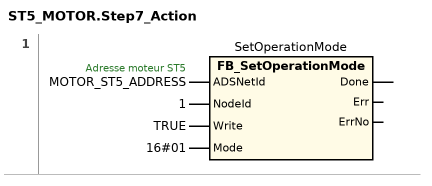
// NETWORK 1
//   MOTOR_ST5_ADDRESS: Adresse moteur ST5
SetOperationMode(ADSNetId := MOTOR_ST5_ADDRESS, NodeId := 1, Write := TRUE, Mode := 16#01); // FB_SetOperationMode
END_ACTION

END_PROGRAM

// ---- POUs/STATIONS/ST1_HT.TcPOU
PROGRAM ST1_HT
VAR
	STEP: INT := 0;
	START_TAMPO_AIR: BOOL;
	TAMPO_AIR: TON;
	JIG_STATUS_R_TRIG: R_TRIG;
	START_TAMPO_CTRLIN: BOOL;
	TAMPO_CTRLIN_TP: TP;
	asdf: TP;
	TAMPO_LIBERATION_TON: TON;
	START_TAMPO_LIBERATION: BOOL;
	TAMPO_SORTIE_VERIN_HAUT_TON: TON;
	START_TAMPO_VERIN_HAUT: BOOL;
	TAMPO_SORTIE_VERIN_ELEC_TON: TON;
	START_TAMPO_VERIN_ELEC: BOOL;
END_VAR

(*******************************************************
*
* Station 1 - Haute Tension
*
*
*********************************************************)
IF NOT(GEMMA.STEP='F1') THEN
	STEP:=0;
END_IF;


CASE STEP OF

0: (*Init*)

	ST1_1V4 := FALSE;
	ST1_1V5 := FALSE;
	
	(*ST1_HT_CTRLIN 	:=FALSE;	(*Prise de contrôle par le PLC*)*)
	ST1_HT_TYPW 	:=FALSE;	(*Type de mesure FALSE: Rigidité dielectrique TRUE:Megomètre*)
	ST1_HT_N0		:=FALSE;	(*Numéro de programme*)
	ST1_HT_N1 		:=FALSE;	(*Numéro de programme*)
	ST1_HT_N2 		:=FALSE;	(*Numéro de programme*)
	ST1_HT_MES_DCH 	:=FALSE;	(*Passage en mesure / décharge FALSE: Décharge TRUE:Mesure*)
	
	FLAGS.ST1_RELEASE_CARRIER := FALSE;
	START_TAMPO_CTRLIN := FALSE;
	START_TAMPO_LIBERATION := FALSE;
	START_TAMPO_VERIN_HAUT := FALSE;
	START_TAMPO_VERIN_ELEC := FALSE;
	
	STEP := STEP + 10;
	
10: (*Attend une palette / flanc montant du status*)

	IF JIG_STATUS_R_TRIG.Q THEN
		STEP := STEP + 10;
	END_IF;
	
20: (*Descend le vérin du dessus*)

	ST1_1V4 := TRUE;
	START_TAMPO_VERIN_HAUT := TRUE;
	STEP := STEP + 10;
	
30: (*Attend vérin dessus sorti*)

	IF TAMPO_SORTIE_VERIN_HAUT_TON.Q THEN
		START_TAMPO_VERIN_HAUT := FALSE;
		STEP := STEP + 10;
	END_IF;

40: (*Sort le vérin électrique*)

	ST1_1V5 := TRUE;
	START_TAMPO_VERIN_ELEC := TRUE;
	STEP := STEP + 10;
	
50: (*Attend vérin électrique sortie*)

	IF TAMPO_SORTIE_VERIN_ELEC_TON.Q THEN
		START_TAMPO_VERIN_ELEC := FALSE;
		STEP := 100;
	END_IF;

	
(**************************************************************************)
100: (*ACtive la prise en main de HT par le PLC et charge le programme*)

	ST1_HT_CTRLIN 	:= TRUE; 	(*active la communication API vers HT*)
	ST1_HT_TYPW 	:= FALSE;	(*Type de mesure FALSE: Rigidité dielectrique TRUE:Megomètre*)
	ST1_HT_N0		:= GETBIT32(inVal32:= INT_TO_DWORD(PUMP_PARAMS.ST1_HT_NO_PROG), bitNo:=0 ) ;	(*Numéro de programme bit 0*)
	ST1_HT_N1 		:= GETBIT32(inVal32:= INT_TO_DWORD(PUMP_PARAMS.ST1_HT_NO_PROG), bitNo:=1 ) ;	(*Numéro de programme bit 1*)
	ST1_HT_N2 		:= GETBIT32(inVal32:= INT_TO_DWORD(PUMP_PARAMS.ST1_HT_NO_PROG), bitNo:=2 ) ;	(*Numéro de programme bit 2*)
	
	STEP := STEP + 10;

110: (*Démarre la mesure*)

	ST1_HT_MES_DCH 	:=TRUE;	(*Passage en mesure / décharge FALSE: Décharge TRUE:Mesure*)
	
	STEP := STEP + 10;	

120: (*Attend début du test HT*)

	IF NOT(ST1_HT_EOT) THEN
		STEP := STEP + 10;
	END_IF;

130: (*Attend la fin du test HT*)

	IF ST1_HT_EOT THEN
		ST1_HT_OK := ST1_HT_PASS;
		STEP := STEP + 10;
	END_IF;
	
140: (*Termine le test*)

	ST1_HT_MES_DCH 	:=FALSE;	(*Passage en mesure / décharge FALSE: Décharge TRUE:Mesure*)
	
	STEP := 300;	

(**************************************************************************)	

300: (*Rentre le vérin électrique*)

	ST1_1V5 := FALSE;
	STEP := STEP + 10;
	
310: (*Monte le vérin du dessus*)

	ST1_1V4 := FALSE;
	STEP := STEP + 10;

320: (*Libère la palette*)
	
	FLAGS.ST1_RELEASE_CARRIER := TRUE;
	STEP := 0;


ELSE
    (*default case*);
END_CASE;

(*FBs*)
TAMPO_SORTIE_VERIN_HAUT_TON(IN:= START_TAMPO_VERIN_HAUT, PT:= TEMPS_SORTIE_VERIN);
TAMPO_SORTIE_VERIN_ELEC_TON(IN:= START_TAMPO_VERIN_ELEC, PT:= TEMPS_SORTIE_VERIN);

TAMPO_CTRLIN_TP(IN:= START_TAMPO_CTRLIN, PT:= T#1S);
TAMPO_LIBERATION_TON(IN:= START_TAMPO_LIBERATION, PT:= T#1S);
JIG_STATUS_R_TRIG(CLK:= CONVEYOR.JIG_ST1.STATUS);
PROG_STEPS.ST1:=STEP;

END_PROGRAM

// ---- POUs/STATIONS/ST2_ASPIRATION.TcPOU
PROGRAM ST2_ASPIRATION
VAR
	STEP: INT := 0;
	JIG_STATUS_R_TRIG: R_TRIG;
	TAMPO_AMORCAGE_TON: TON;
	START_TAMPO_AMORCAGE: BOOL;
	TAMPO_MESURE_TON: TON;
	START_TAMPO_MESURE: BOOL;
	TAMPO_SORTIE_VERIN_HAUT_TON: TON;
	START_TAMPO_VERIN_HAUT: BOOL;
	TAMPO_SORTIE_VERIN_BAS_TON: TON;
	START_TAMPO_VERIN_BAS: BOOL;
	TAMPO_SORTIE_VERIN_ELEC_TON: TON;
	START_TAMPO_VERIN_ELEC: BOOL;
	START_TAMPO_MESURE_PERTES: BOOL;
	TAMPO_MESURE_PERTES_TON: TON;
END_VAR

(*******************************************************
*
* Station 2 - Aspiration
*
*
*********************************************************)
IF NOT(GEMMA.STEP='F1') THEN
	STEP:=0;
END_IF;


CASE STEP OF

0: (*Init*)

	ST2_2V4 := FALSE;
	ST2_2V5 := FALSE;
	ST2_2V6 := FALSE;
	ST2_2V7 := FALSE;
	ST2_2V8 := FALSE;
	
	FLAGS.ST2_RELEASE_CARRIER := FALSE;
	START_TAMPO_AMORCAGE := FALSE;
	START_TAMPO_MESURE := FALSE;
	START_TAMPO_VERIN_ELEC := FALSE;
	START_TAMPO_VERIN_HAUT := FALSE;
	START_TAMPO_VERIN_BAS := FALSE;
	
	STEP := STEP + 10;
	
10: (*Attend une palette / flanc montant du status*)

	IF JIG_STATUS_R_TRIG.Q THEN
		STEP := STEP + 10;
	END_IF;
	
20: (*Descend le vérin du dessus*)

	ST2_2V4 := TRUE;
	START_TAMPO_VERIN_HAUT := TRUE;
	STEP := STEP + 10;
	
30: (*Attend vérin dessus sorti*)

	IF TAMPO_SORTIE_VERIN_HAUT_TON.Q THEN
		START_TAMPO_VERIN_HAUT := FALSE;
		STEP := STEP + 10;
	END_IF;

40: (*Monte le vérin du dessous*)

	ST2_2V5 := TRUE;
	START_TAMPO_VERIN_BAS := TRUE;
	STEP := STEP + 10;
	
50: (*Attend vérin dessus sorti*)

	IF TAMPO_SORTIE_VERIN_BAS_TON.Q THEN
		START_TAMPO_VERIN_BAS := FALSE;
		STEP := STEP + 10;
	END_IF;
	
60: (*Sort le vérin électrique*)

	ST2_2V6 := TRUE;
	IF PUMP_PARAMS.GEN_BYPASS THEN
		ST2_2V7 := TRUE;
	END_IF
	START_TAMPO_VERIN_ELEC := TRUE;
	STEP := STEP + 10;
	
70: (*Attend vérin électrique sortie*)

	IF TAMPO_SORTIE_VERIN_ELEC_TON.Q THEN
		START_TAMPO_VERIN_ELEC := FALSE;
		STEP := STEP + 10;
	END_IF;

80: (*Allume la pompe*)

	IF PUMP_PARAMS.ST2_CONTRE_PRESSION THEN (*ouvre la vanne de contre pression d'air si nécessaire*)
		ST2_2V8:=TRUE;
	END_IF;
	
	ST2_POWER := TRUE;
	STEP := 100;
	
(**************************************************************************)
100: (*Démarre la tampo pour l'amorcage*)

	START_TAMPO_AMORCAGE := TRUE;
	STEP := STEP + 10;
	
110: (*Attend fin tampo amorcage*)

	IF TAMPO_AMORCAGE_TON.Q THEN
		START_TAMPO_AMORCAGE := FALSE;
		STEP := STEP + 10;
	END_IF;
	
120: (*Démarre la tampo pour la mesure de pression*)

	START_TAMPO_MESURE := TRUE;
	STEP := STEP + 10;
	
130: (*Attend fin tampo mesure - MESURE EN COURT*)

	IF TAMPO_MESURE_TON.Q THEN
		START_TAMPO_MESURE := FALSE;
		ST2_2V8:=FALSE; (*ferme la vanne de contre pression d'air*)
		STEP := STEP + 10;
	END_IF;
	
140: (*Démarre la tampo pour la mesure de la tenue aspiration*)

	START_TAMPO_MESURE_PERTES := TRUE;
	ST2_POWER := FALSE;
	STEP := STEP + 10;
	
150: (*Attend fin tampo mesure - MESURE EN COURT tenue aspiration*)

	IF TAMPO_MESURE_PERTES_TON.Q THEN
		START_TAMPO_MESURE_PERTES := FALSE;
		ST2_2V8:=FALSE; (*ferme la vanne de contre pression d'air*)
		STEP := 300;
	END_IF;
	

(**************************************************************************)	

300: (*Rentre le vérin électrique*)

	ST2_2V6 := FALSE;
	ST2_2V7 := TRUE;
	STEP := STEP + 10;
	
310: (*Descend le vérin du dessous*)

	ST2_2V5 := FALSE;
	STEP := STEP + 10;
	
320: (*Monte le vérin du dessus*)

	ST2_2V4 := FALSE;
	STEP := STEP + 10;

330: (*Libère la palette*)

	FLAGS.ST2_RELEASE_CARRIER := TRUE;
	STEP := 0;


ELSE
    (*default case*);
END_CASE;

(*FBs*)
TAMPO_SORTIE_VERIN_HAUT_TON(IN:= START_TAMPO_VERIN_HAUT, PT:= TEMPS_SORTIE_VERIN);
TAMPO_SORTIE_VERIN_BAS_TON(IN:= START_TAMPO_VERIN_BAS, PT:= TEMPS_SORTIE_VERIN);
TAMPO_SORTIE_VERIN_ELEC_TON(IN:= START_TAMPO_VERIN_ELEC, PT:= TEMPS_SORTIE_VERIN);

TAMPO_AMORCAGE_TON(IN:= START_TAMPO_AMORCAGE, PT:= PUMP_PARAMS.ST6_TEMPS_POMPAGE);
TAMPO_MESURE_TON(IN:= START_TAMPO_MESURE, PT:= PUMP_PARAMS.ST6_TEMPS_MESURE);
TAMPO_MESURE_PERTES_TON(IN:= START_TAMPO_MESURE_PERTES, PT:= PUMP_PARAMS.ST2_TEMPS_MESURE_PERTE_PRESSION);
JIG_STATUS_R_TRIG(CLK:= CONVEYOR.JIG_ST2.STATUS);
PROG_STEPS.ST2:=STEP;

END_PROGRAM

// ---- POUs/STATIONS/ST3_ETANCHEITE.TcPOU
PROGRAM ST3_ETANCHEITE
VAR
	STEP: INT := 0;
	JIG_STATUS_R_TRIG: R_TRIG;
	START_TAMPO_MISE_SOUS_PRESSION: BOOL;
	TAMPO_MISE_SOUS_PRESSION: TON;
	START_TAMPO_STABILISATION: BOOL;
	TAMPO_STABILISATION: TON;
	START_TAMPO_MESURE: BOOL;
	TAMPO_MESURE: TON;
	PRESSION_DEBUT: REAL;
	PRESSION_FIN: REAL;
	TAMPO_SORTIE_VERIN_HAUT_TON: TON;
	START_TAMPO_VERIN_HAUT: BOOL;
	TAMPO_SORTIE_VERIN_BAS_TON: TON;
	START_TAMPO_VERIN_BAS: BOOL;
	TAMPO_DEPRESSION_TON: TON;
	START_TAMPO_DEPRESSION: BOOL;
	PRESSION_DEBUT_ABS: REAL;
END_VAR

(*******************************************************
*
* Station 3 - Etanchéité
*
*
*********************************************************)
IF NOT(GEMMA.STEP='F1') THEN
	STEP:=0;
END_IF;


CASE STEP OF

0: (*Init*)

	ST3_3V4 := FALSE;
	ST3_3V5 := FALSE;
	ST3_3V10 := FALSE;
	ST3_3V11 := FALSE;
	ST3_3V12 := TRUE;
	
	FLAGS.ST3_RELEASE_CARRIER := FALSE;
	
	START_TAMPO_MISE_SOUS_PRESSION := FALSE;
	START_TAMPO_STABILISATION := FALSE;
	START_TAMPO_MESURE := FALSE;
	START_TAMPO_VERIN_HAUT := FALSE;
	START_TAMPO_VERIN_BAS := FALSE;
	START_TAMPO_DEPRESSION := FALSE;

	
	STEP := STEP + 10;
	
10: (*Attend une palette / flanc montant du status*)

	IF JIG_STATUS_R_TRIG.Q THEN
		STEP := STEP + 10;
	END_IF;
	
20: (*Descend le vérin du dessus*)

	ST3_3V4 := TRUE;
	START_TAMPO_VERIN_HAUT := TRUE;
	STEP := STEP + 10;
	
30: (*Attend vérin dessus sorti*)

	IF TAMPO_SORTIE_VERIN_HAUT_TON.Q THEN
		START_TAMPO_VERIN_HAUT :=FALSE;
		STEP := STEP + 10;
	END_IF;

40: (*Monte le vérin du dessous*)

	ST3_3V5 := TRUE;
	IF PUMP_PARAMS.GEN_BYPASS THEN
		ST3_3V7 := TRUE;
	END_IF
	START_TAMPO_VERIN_BAS := TRUE;
	STEP := STEP + 10;
	
50: (*Attend vérin dessus sorti*)

	IF TAMPO_SORTIE_VERIN_BAS_TON.Q THEN
		START_TAMPO_VERIN_BAS := FALSE;
		STEP := 100;
	END_IF;
	
	
(**************************************************************************)
100: (*Mise sous pression de la cartouche*)

	ST3_3V10 := TRUE;
	ST3_3V11 := FALSE;
	ST3_3V12 := TRUE;
	
	START_TAMPO_MISE_SOUS_PRESSION := TRUE;
	
	STEP := STEP + 10;
	
	
110: (*Tampo pour la mise sous pression de la cartouche*)

	IF TAMPO_MISE_SOUS_PRESSION.Q THEN
		START_TAMPO_MISE_SOUS_PRESSION := FALSE;
		STEP := STEP + 10;
	END_IF;

120: (*Start stabilisation*)

	START_TAMPO_STABILISATION := TRUE;
	ST3_3V10 := FALSE;
	
	STEP := STEP + 10;	

130: (*Tampo pour la stabilisation de la pression dans la cartouche*)

	IF TAMPO_STABILISATION.Q THEN
		START_TAMPO_STABILISATION := FALSE;
		STEP := STEP + 10;
	END_IF;
	
140: (*Start mesure*)

	START_TAMPO_MESURE := TRUE;
	ST3_3V12 := FALSE;
	PRESSION_DEBUT := ST3_PRESSION; (* Mesure de la pression différentielle au début du test *)
	
	STEP := STEP + 10;	

150: (*Tampo pour la mesure du delta P*)

	IF TAMPO_MESURE.Q THEN
		START_TAMPO_MESURE := FALSE;
		PRESSION_FIN := ST3_PRESSION; (* Mesure de la pression à la fin du test *)
		ST3_PRESSION_FIN_ABS := ST3_PRESSION_ABS; (* Mesure de la pression par rapport à l'atmosphère à la fin du test *)
		ST3_DELTA_P := PRESSION_FIN - PRESSION_DEBUT; (* Calcule de la chutte de pression *)
		STEP := STEP + 10;
	END_IF;
	
160: (*Fin mesure, dépressiorisation de la cartouche*)

	ST3_3V10 := FALSE;
	ST3_3V11 := TRUE;
	ST3_3V12 := TRUE;
	
	START_TAMPO_DEPRESSION := TRUE;
	
	STEP := STEP + 10;

170: (*Tampo dépression de cartouche*)

	IF TAMPO_DEPRESSION_TON.Q THEN
		START_TAMPO_DEPRESSION := FALSE;
		STEP := 300;
	END_IF;	
	
	

(**************************************************************************)	

300: (*Descend le vérin du dessous*)

	ST3_3V5 := FALSE;
	ST3_3V7 := FALSE;
	STEP := STEP + 10;
	
310: (*Monte le vérin du dessus*)

	ST3_3V4 := FALSE;
	STEP := STEP + 10;

320: (*Libère la palette*)

	FLAGS.ST3_RELEASE_CARRIER := TRUE;
	STEP := 0;


ELSE
    (*default case*);
END_CASE;

(*FBs*)

TAMPO_SORTIE_VERIN_HAUT_TON(IN:= START_TAMPO_VERIN_HAUT, PT:= TEMPS_SORTIE_VERIN);
TAMPO_SORTIE_VERIN_BAS_TON(IN:= START_TAMPO_VERIN_BAS, PT:= TEMPS_SORTIE_VERIN);

TAMPO_DEPRESSION_TON(IN:= START_TAMPO_DEPRESSION, PT:= T#2S);
TAMPO_MISE_SOUS_PRESSION(IN:= START_TAMPO_MISE_SOUS_PRESSION, PT:= PUMP_PARAMS.ST3_TEMPS_MISE_SOUS_PRESSION);
TAMPO_STABILISATION(IN:= START_TAMPO_STABILISATION, PT:= PUMP_PARAMS.ST3_TEMPS_STABILISATION);
TAMPO_MESURE(IN:= START_TAMPO_MESURE, PT:= PUMP_PARAMS.ST3_TEMPS_MESURE);
JIG_STATUS_R_TRIG(CLK:= CONVEYOR.JIG_ST3.STATUS);
PROG_STEPS.ST3:=STEP;

END_PROGRAM

// ---- POUs/STATIONS/ST4_DEBIT_PETIT.TcPOU
PROGRAM ST4_DEBIT_PETIT
VAR
	STEP: INT := 0;
	JIG_STATUS_R_TRIG: R_TRIG;
	START_TAMPO_AMORCAGE: BOOL;
	TAMPO_AMORCAGE_TON: TON;
	START_TAMPO_REGLAGE: BOOL;
	TAMPO_REGLAGE_TON: TON;
	START_TAMPO_MESURE_DEBIT: BOOL;
	TAMPO_MESURE_DEBIT_TON: TON;
	START_TAMPO_VIDANGE: BOOL;
	TAMPO_VIDANGE_TON: TON;
	START_TAMPO_MESURE_DEBIT_MAX: BOOL;
	TAMPO_MESURE_DEBIT_MAX_TON: TON;
	POIDS_QMAX_DEBUT: REAL;
	POIDS_Q_DEBUT: REAL;
	P_ERREUR: REAL;
	START_TAMPO_PRESSION: BOOL;
	TAMPO_PRESSION_TON: TON;
		TAMPO_SORTIE_VERIN_HAUT_TON: TON;
	START_TAMPO_VERIN_HAUT: BOOL;
	TAMPO_SORTIE_VERIN_BAS_TON: TON;
	START_TAMPO_VERIN_BAS: BOOL;
	TAMPO_SORTIE_VERIN_ELEC_TON: TON;
	START_TAMPO_VERIN_ELEC: BOOL;
END_VAR

(*******************************************************
*
* Station 4 - Petits débits
*
*
*********************************************************)
IF NOT(GEMMA.STEP='F1') THEN
	STEP:=0;
END_IF;


CASE STEP OF

0: (*Init*)

	ST4_4V4 := FALSE;
	ST4_4V5 := FALSE;
	ST4_4V6 := FALSE;
	ST4_4V7 := FALSE;

	ST4_4V10 := FALSE;
	ST4_4V12 := FALSE;
	ST4_4V13 := FALSE;
	
	
	FLAGS.ST4_RELEASE_CARRIER := FALSE;
	START_TAMPO_AMORCAGE := FALSE;
	START_TAMPO_MESURE_DEBIT:= FALSE;
	START_TAMPO_MESURE_DEBIT_MAX:= FALSE;
	START_TAMPO_VIDANGE:= FALSE;
	START_TAMPO_REGLAGE:= FALSE;
	START_TAMPO_PRESSION:= FALSE;
	START_TAMPO_VERIN_ELEC := FALSE;
	START_TAMPO_VERIN_HAUT := FALSE;
	START_TAMPO_VERIN_BAS := FALSE;
	
	
	STEP := STEP + 10;
	
10: (*Attend une palette / flanc montant du status*)

	IF JIG_STATUS_R_TRIG.Q THEN
		STEP := STEP + 10;
	END_IF;
	
20: (*Descend le vérin du dessus*)

	ST4_4V4 := TRUE;
	START_TAMPO_VERIN_HAUT := TRUE;
	POIDS_QMAX_DEBUT	:= 0;	(*Met à 0 les différentes variables pour le calcul et résultat des débits*)
	POIDS_Q_DEBUT		:= 0;
	ST4_Q				:= 0;
	ST4_QMAX			:= 0;
	STEP := STEP + 10;
	
30: (*Attend vérin dessus sorti*)

	IF TAMPO_SORTIE_VERIN_HAUT_TON.Q THEN
		START_TAMPO_VERIN_HAUT := FALSE;
		STEP := STEP + 10;
	END_IF;

40: (*Monte le vérin du dessous*)

	ST4_4V5 := TRUE;
	START_TAMPO_VERIN_BAS := TRUE;
	STEP := STEP + 10;
	
50: (*Attend vérin dessus sorti*)

	IF TAMPO_SORTIE_VERIN_BAS_TON.Q THEN
		START_TAMPO_VERIN_BAS := FALSE;
		STEP := STEP + 10;
	END_IF;
	
60: (*Sort le vérin électrique*)

	ST4_4V6 := TRUE;
	IF PUMP_PARAMS.GEN_BYPASS THEN
		ST4_4V7 := TRUE;
	END_IF
	START_TAMPO_VERIN_ELEC := TRUE;
	STEP := STEP + 10;
	
70: (*Attend vérin électrique sortie*)

	IF TAMPO_SORTIE_VERIN_ELEC_TON.Q THEN
		START_TAMPO_VERIN_ELEC := FALSE;
		STEP := STEP + 10;
	END_IF;
	
80: (*Si la balance est trop pleine, attend qu'elle soit vidée suffisament avant d'allumer la pompe*)
	
	IF ST4_POIDS<BALANCE_POIDS_LIMITE THEN
		STEP:=STEP + 10;
	END_IF
		
90: (*Allume la pompe*)

	ST4_POWER := TRUE;
	ST4_4V10 := TRUE;
	ST4_4V13 := TRUE;
	STEP := 100;
	
	
(**************************************************************************)
100: (*Démarre la tampo pour l'amorcage*)

	START_TAMPO_AMORCAGE := TRUE;
	STEP := STEP + 10;
	
110: (*Attend fin tampo amorcage*)

	IF TAMPO_AMORCAGE_TON.Q THEN
		START_TAMPO_AMORCAGE := FALSE;
		STEP := STEP + 10;
	END_IF;
	
120: (*Démarre la tampo pour la mesure de Qmax*)

	START_TAMPO_MESURE_DEBIT_MAX := TRUE;
	POIDS_QMAX_DEBUT := ST4_POIDS;
	STEP := STEP + 10;
	
130: (*Attend fin tampo mesure de Qmax ***********************************************************)
	IF TAMPO_MESURE_DEBIT_MAX_TON.Q THEN
		ST4_QMAX := CONVERT_MASS_TO_FLOW(ST4_POIDS - POIDS_QMAX_DEBUT, PUMP_PARAMS.ST45_TEMPS_MESURE_DEBIT_MAX);(*Calcul du débit max*)
		
		QMAX_ARRAY[INDEX_QMAX_ARRAY]:=ST4_QMAX; (*Array des derniers résultats*)
		INDEX_QMAX_ARRAY := INDEX_QMAX_ARRAY+1;
		
		START_TAMPO_MESURE_DEBIT_MAX := FALSE;
		ST4_4V12 := TRUE;
		ST4_4V13 := FALSE;
		STEP := STEP + 10;
	END_IF;
	
140: (*Démarre la tampo pour la mise sous pression*)

	START_TAMPO_PRESSION := TRUE;
	STEP := STEP + 10;
	
150: (*Attend fin tampo mise sous pression*)

	IF TAMPO_PRESSION_TON.Q THEN
		START_TAMPO_PRESSION := FALSE;
		STEP := STEP + 10;
	END_IF;
	
160: (*Démarre la tampo pour le réglage*)

	START_TAMPO_REGLAGE := TRUE;
	STEP := STEP + 10;
	
170: (*Attend fin tampo réglage*)

(*Réglage pression**********************************************)
PRESSURE_REGULATOR_ST4(
GEMMA				:= GEMMA.STEP,
COURANT				:= ST4_COURANT, 
PRESSION_CONSIGNE	:= PUMP_PARAMS.ST45_PRESSION_CONSIGNE, 
PRESSION_MESURE		:= ST4_PRESSURE_FILTERED,
MOTOR_POSITION_MAX	:= MOTOR_ST4_POSITION_MAX,
MOTOR_INITIAL_POSITION := MOTOR_ST4_INITIAL_POS,
MOTOR_POSITION		=> FLAGS.MOTOR_ST4_POSITION
);
	

	IF TAMPO_REGLAGE_TON.Q THEN
		START_TAMPO_REGLAGE := FALSE;
		STEP := STEP + 10;
	END_IF;
	
180: (*Démarre la tampo pour la mesure de debit*************************************************)

	START_TAMPO_MESURE_DEBIT := TRUE;
	POIDS_Q_DEBUT := ST4_POIDS;
	STEP := STEP + 10;

	
190: (*Attend fin tampo amorcage - MESURE EN COURT*)

(*Réglage pression***********************************************)
PRESSURE_REGULATOR_ST4( 
GEMMA				:= GEMMA.STEP,
COURANT				:= ST4_COURANT, 
PRESSION_CONSIGNE	:= PUMP_PARAMS.ST45_PRESSION_CONSIGNE, 
PRESSION_MESURE		:= ST4_PRESSURE_FILTERED,
MOTOR_POSITION_MAX	:= MOTOR_ST4_POSITION_MAX,
MOTOR_INITIAL_POSITION := MOTOR_ST4_INITIAL_POS,
MOTOR_POSITION		=> FLAGS.MOTOR_ST4_POSITION
);

	IF TAMPO_MESURE_DEBIT_TON.Q THEN
		ST4_Q := CONVERT_MASS_TO_FLOW(ST4_POIDS - POIDS_Q_DEBUT, PUMP_PARAMS.ST45_TEMPS_MESURE_DEBIT);(*Calcul du débit de travail*)
		
		Q_ARRAY[INDEX_Q_ARRAY]:=ST4_Q; (*Array des derniers résultats*)
		INDEX_Q_ARRAY := INDEX_Q_ARRAY+1;
		
		START_TAMPO_MESURE_DEBIT := FALSE;
		STEP := 300;
	END_IF;
	
	

(**************************************************************************)	

300: (*Descend le vérin du dessous*)

	ST4_4V5 := FALSE;
	ST4_4V10 := FALSE;	(* ferme la vanne avant la pompe*)
	ST4_4V12 := FALSE;
	ST4_4V13 := TRUE;
	STEP := STEP + 10;

310: (*Démarre la tampo de vidange de la pompe*)

	START_TAMPO_VIDANGE := TRUE;
	STEP := STEP + 10;
	
320: (*Attend fin tampo amorcage*)

	IF TAMPO_VIDANGE_TON.Q THEN
		START_TAMPO_VIDANGE := FALSE;
		ST4_4V13 := FALSE;
		ST4_POWER := FALSE;
		STEP := STEP + 10;
	END_IF;

330: (*Rentre le vérin électrique*)

	ST4_4V6 := FALSE;
	ST4_4V7 := FALSE;
	STEP := STEP + 10;
	
	
340: (*Monte le vérin du dessus*)

	ST4_4V4 := FALSE;
	STEP := STEP + 10;

350: (*Libère la palette*)

	FLAGS.ST4_RELEASE_CARRIER := TRUE;
	STEP := 0;


ELSE
    (*default case*);
END_CASE;

(*FBs*)
TAMPO_SORTIE_VERIN_HAUT_TON(IN:= START_TAMPO_VERIN_HAUT, PT:= TEMPS_SORTIE_VERIN);
TAMPO_SORTIE_VERIN_BAS_TON(IN:= START_TAMPO_VERIN_BAS, PT:= TEMPS_SORTIE_VERIN);
TAMPO_SORTIE_VERIN_ELEC_TON(IN:= START_TAMPO_VERIN_ELEC, PT:= TEMPS_SORTIE_VERIN);

TAMPO_AMORCAGE_TON(IN:= START_TAMPO_AMORCAGE, PT:= PUMP_PARAMS.ST45_TEMPS_POMPAGE);
TAMPO_REGLAGE_TON(IN:= START_TAMPO_REGLAGE, PT:= PUMP_PARAMS.ST45_TEMPS_REGLAGE_PRESSION);
TAMPO_VIDANGE_TON(IN:= START_TAMPO_VIDANGE, PT:= TEMPS_VIDANGE_POMPE);
TAMPO_PRESSION_TON(IN:= START_TAMPO_PRESSION, PT:= TEMPS_CHANGEMENT_PRESSION);
TAMPO_MESURE_DEBIT_TON(IN:= START_TAMPO_MESURE_DEBIT, PT:= PUMP_PARAMS.ST45_TEMPS_MESURE_DEBIT);
TAMPO_MESURE_DEBIT_MAX_TON(IN:= START_TAMPO_MESURE_DEBIT_MAX, PT:= PUMP_PARAMS.ST45_TEMPS_MESURE_DEBIT_MAX);
JIG_STATUS_R_TRIG(CLK:= CONVEYOR.JIG_ST4.STATUS);
PROG_STEPS.ST4:=STEP;

END_PROGRAM

// ---- POUs/Functions/CONVERT_MASS_TO_FLOW.TcPOU
FUNCTION CONVERT_MASS_TO_FLOW : REAL
VAR_INPUT
	Mass:REAL; (*in gramme*)
	Delay:TIME; (*in ms*)
END_VAR
VAR
END_VAR

CONVERT_MASS_TO_FLOW:=Mass/TIME_TO_DWORD(Delay)*60*60;

END_FUNCTION

// ---- POUs/STATIONS/ST5_GRAND_PETIT.TcPOU
PROGRAM ST5_GRAND_PETIT
VAR
	STEP: INT := 0;
	JIG_STATUS_R_TRIG: R_TRIG;
	START_TAMPO_AMORCAGE: BOOL;
	TAMPO_AMORCAGE_TON: TON;
	START_TAMPO_REGLAGE: BOOL;
	TAMPO_REGLAGE_TON: TON;
	START_TAMPO_MESURE_DEBIT: BOOL;
	TAMPO_MESURE_DEBIT_TON: TON;
	START_TAMPO_VIDANGE: BOOL;
	TAMPO_VIDANGE_TON: TON;
	START_TAMPO_MESURE_DEBIT_MAX: BOOL;
	TAMPO_MESURE_DEBIT_MAX_TON: TON;
	POIDS_QMAX_DEBUT: REAL;
	POIDS_Q_DEBUT: REAL;
	P_ERREUR: REAL;
	START_TAMPO_PRESSION: BOOL;
	TAMPO_PRESSION_TON: TON;
	TAMPO_SORTIE_VERIN_HAUT_TON: TON;
	START_TAMPO_VERIN_HAUT: BOOL;
	TAMPO_SORTIE_VERIN_BAS_TON: TON;
	START_TAMPO_VERIN_BAS: BOOL;
	TAMPO_SORTIE_VERIN_ELEC_TON: TON;
	START_TAMPO_VERIN_ELEC: BOOL;
	TAMPO_RENTREE_VERIN_HAUT_TON: TON;
	START_TAMPO_RENTREE_VERIN_HAUT: BOOL;
END_VAR

(*******************************************************
*
* Station 5 - Grands débits
*
*
*********************************************************)
IF NOT(GEMMA.STEP='F1') THEN
	STEP:=0;
END_IF;


CASE STEP OF

0: (*Init*)

	ST5_5V4 := FALSE;
	ST5_5V5 := FALSE;
	ST5_5V6 := FALSE;

	ST5_5V10 := FALSE;
	ST5_5V12 := FALSE;
	ST5_5V13 := FALSE;
	
	
	FLAGS.ST5_RELEASE_CARRIER := FALSE;
	START_TAMPO_AMORCAGE := FALSE;
	START_TAMPO_MESURE_DEBIT:= FALSE;
	START_TAMPO_MESURE_DEBIT_MAX:= FALSE;
	START_TAMPO_VIDANGE:= FALSE;
	START_TAMPO_REGLAGE:= FALSE;
	START_TAMPO_PRESSION:= FALSE;
	START_TAMPO_VERIN_ELEC := FALSE;
	START_TAMPO_VERIN_HAUT := FALSE;
	START_TAMPO_VERIN_BAS := FALSE;
	
	
	STEP := STEP + 10;
	
10: (*Attend une palette / flanc montant du status*)

	IF JIG_STATUS_R_TRIG.Q THEN
		STEP := STEP + 10;
	END_IF;
	
20: (*Descend le vérin du dessus*)

	ST5_5V4 := TRUE;
	START_TAMPO_VERIN_HAUT := TRUE;
	POIDS_QMAX_DEBUT	:= 0;	(*Met à 0 les différentes variables pour le calcul et résultat des débits*)
	POIDS_Q_DEBUT		:= 0;
	ST5_Q				:= 0;
	ST5_QMAX			:= 0;
	STEP := STEP + 10;
	
30: (*Attend vérin dessus sorti*)

	IF TAMPO_SORTIE_VERIN_HAUT_TON.Q THEN
		START_TAMPO_VERIN_HAUT := FALSE;
		STEP := STEP + 10;
	END_IF;

40: (*Monte le vérin du dessous*)

	ST5_5V5 := TRUE;
	START_TAMPO_VERIN_BAS := TRUE;
	STEP := STEP + 10;
	
50: (*Attend vérin dessus sorti*)

	IF TAMPO_SORTIE_VERIN_BAS_TON.Q THEN
		START_TAMPO_VERIN_BAS := FALSE;
		STEP := STEP + 10;
	END_IF;
	
60: (*Sort le vérin électrique*)

	ST5_5V6 := TRUE;
	START_TAMPO_VERIN_ELEC := TRUE;
	STEP := STEP + 10;
	
70: (*Attend vérin électrique sortie*)

	IF TAMPO_SORTIE_VERIN_ELEC_TON.Q THEN
		START_TAMPO_VERIN_ELEC := FALSE;
		STEP := STEP + 10;
	END_IF;

80: (*Si la balance est trop pleine, attend qu'elle soit vidée suffisament avant d'allumer la pompe*)
	
IF ST5_POIDS<BALANCE_POIDS_LIMITE THEN
	STEP:=STEP + 10;
END_IF
	
90: (*Allume la pompe*)

	ST5_POWER := TRUE;
	ST5_5V10 := TRUE;
	ST5_5V13 := TRUE;
	STEP := 100;
	
	
(**************************************************************************)
100: (*Démarre la tampo pour l'amorcage*)

	START_TAMPO_AMORCAGE := TRUE;
	STEP := STEP + 10;
	
110: (*Attend fin tampo amorcage*)

	IF TAMPO_AMORCAGE_TON.Q THEN
		START_TAMPO_AMORCAGE := FALSE;
		STEP := STEP + 10;
	END_IF;
	
120: (*Démarre la tampo pour la mesure de Qmax*)

	START_TAMPO_MESURE_DEBIT_MAX := TRUE;
	POIDS_QMAX_DEBUT := ST5_POIDS;
	STEP := STEP + 10;
	
130: (*Attend fin tampo mesure de Qmax ***********************************************************)
	IF TAMPO_MESURE_DEBIT_MAX_TON.Q THEN
		ST5_QMAX := CONVERT_MASS_TO_FLOW(ST5_POIDS - POIDS_QMAX_DEBUT, PUMP_PARAMS.ST45_TEMPS_MESURE_DEBIT_MAX);(*Calcul du débit max*)
		
		QMAX5_ARRAY[INDEX_QMAX5_ARRAY]:=ST5_QMAX; (*Array des derniers résultats*)
		INDEX_QMAX5_ARRAY := INDEX_QMAX5_ARRAY+1;
		
		START_TAMPO_MESURE_DEBIT_MAX := FALSE;
		ST5_5V12 := TRUE;
		ST5_5V13 := FALSE;
		STEP := STEP + 10;
	END_IF;
	
140: (*Démarre la tampo pour la mise sous pression*)

	START_TAMPO_PRESSION := TRUE;
	STEP := STEP + 10;
	
150: (*Attend fin tampo mise sous pression*)

	IF TAMPO_PRESSION_TON.Q THEN
		START_TAMPO_PRESSION := FALSE;
		STEP := STEP + 10;
	END_IF;
	
160: (*Démarre la tampo pour le réglage*)

	START_TAMPO_REGLAGE := TRUE;
	STEP := STEP + 10;
	
170: (*Attend fin tampo réglage*)

(*Réglage pression**********************************************)
PRESSURE_REGULATOR_ST5(
GEMMA				:= GEMMA.STEP,
COURANT				:= ST5_COURANT, 
PRESSION_CONSIGNE	:= PUMP_PARAMS.ST45_PRESSION_CONSIGNE, 
PRESSION_MESURE		:= ST5_PRESSURE_FILTERED,
MOTOR_POSITION_MAX	:= MOTOR_ST5_POSITION_MAX,
MOTOR_INITIAL_POSITION := MOTOR_ST5_INITIAL_POS,
MOTOR_POSITION		=> FLAGS.MOTOR_ST5_POSITION
);
	

	IF TAMPO_REGLAGE_TON.Q THEN
		START_TAMPO_REGLAGE := FALSE;
		STEP := STEP + 10;
	END_IF;
	
180: (*Démarre la tampo pour la mesure de debit*************************************************)

	START_TAMPO_MESURE_DEBIT := TRUE;
	POIDS_Q_DEBUT := ST5_POIDS;
	STEP := STEP + 10;

	
190: (*Attend fin tampo amorcage - MESURE EN COURT*)

(*Réglage pression***********************************************)
PRESSURE_REGULATOR_ST5( 
GEMMA				:= GEMMA.STEP,
COURANT				:= ST5_COURANT, 
PRESSION_CONSIGNE	:= PUMP_PARAMS.ST45_PRESSION_CONSIGNE, 
PRESSION_MESURE		:= ST5_PRESSURE_FILTERED,
MOTOR_POSITION_MAX	:= MOTOR_ST5_POSITION_MAX,
MOTOR_INITIAL_POSITION := MOTOR_ST5_INITIAL_POS,
MOTOR_POSITION		=> FLAGS.MOTOR_ST5_POSITION
);

	IF TAMPO_MESURE_DEBIT_TON.Q THEN
		ST5_Q := CONVERT_MASS_TO_FLOW(ST5_POIDS - POIDS_Q_DEBUT, PUMP_PARAMS.ST45_TEMPS_MESURE_DEBIT);(*Calcul du débit de travail*)
		
		Q5_ARRAY[INDEX_Q5_ARRAY]:=ST5_Q; (*Array des derniers résultats*)
		INDEX_Q5_ARRAY := INDEX_Q5_ARRAY+1;
		
		START_TAMPO_MESURE_DEBIT := FALSE;
		STEP := 300;
	END_IF;
	
	

(**************************************************************************)	

300: (*Descend le vérin du dessous*)

	ST5_5V5 := FALSE;
	ST5_5V10 := FALSE;	(* ferme la vanne avant la pompe*)
	ST5_5V12 := FALSE;
	ST5_5V13 := TRUE;
	STEP := STEP + 10;

310: (*Démarre la tampo de vidange de la pompe*)

	START_TAMPO_VIDANGE := TRUE;
	STEP := STEP + 10;
	
320: (*Attend fin tampo amorcage*)

	IF TAMPO_VIDANGE_TON.Q THEN
		START_TAMPO_VIDANGE := FALSE;
		ST5_5V13 := FALSE;
		ST5_POWER := FALSE;
		STEP := STEP + 10;
	END_IF;

330: (*Rentre le vérin électrique*)

	ST5_5V6 := FALSE;
	STEP := STEP + 10;
	
	
340: (*Monte le vérin du dessus*)

	ST5_5V4 := FALSE;
	START_TAMPO_RENTREE_VERIN_HAUT:=TRUE;
	STEP := STEP + 10;
	
350: (*Attend vérin du dessus rentré légèrement (pour éviter que la pompe tape contre)*)

	IF TAMPO_RENTREE_VERIN_HAUT_TON.Q THEN
		START_TAMPO_RENTREE_VERIN_HAUT := FALSE;
		STEP := STEP + 10;
	END_IF;

360: (*Libère la palette*)

	FLAGS.ST5_RELEASE_CARRIER := TRUE;
	STEP := 0;


ELSE
    (*default case*);
END_CASE;

(*FBs*)
TAMPO_SORTIE_VERIN_HAUT_TON(IN:= START_TAMPO_VERIN_HAUT, PT:= TEMPS_SORTIE_VERIN);
TAMPO_SORTIE_VERIN_BAS_TON(IN:= START_TAMPO_VERIN_BAS, PT:= TEMPS_SORTIE_VERIN);
TAMPO_SORTIE_VERIN_ELEC_TON(IN:= START_TAMPO_VERIN_ELEC, PT:= TEMPS_SORTIE_VERIN);
TAMPO_RENTREE_VERIN_HAUT_TON(IN:= START_TAMPO_RENTREE_VERIN_HAUT, PT:= TEMPS_RENTREE_VERIN);

TAMPO_AMORCAGE_TON(IN:= START_TAMPO_AMORCAGE, PT:= PUMP_PARAMS.ST45_TEMPS_POMPAGE);
TAMPO_REGLAGE_TON(IN:= START_TAMPO_REGLAGE, PT:= PUMP_PARAMS.ST45_TEMPS_REGLAGE_PRESSION);
TAMPO_VIDANGE_TON(IN:= START_TAMPO_VIDANGE, PT:= TEMPS_VIDANGE_POMPE);
TAMPO_PRESSION_TON(IN:= START_TAMPO_PRESSION, PT:= TEMPS_CHANGEMENT_PRESSION);
TAMPO_MESURE_DEBIT_TON(IN:= START_TAMPO_MESURE_DEBIT, PT:= PUMP_PARAMS.ST45_TEMPS_MESURE_DEBIT);
TAMPO_MESURE_DEBIT_MAX_TON(IN:= START_TAMPO_MESURE_DEBIT_MAX, PT:= PUMP_PARAMS.ST45_TEMPS_MESURE_DEBIT_MAX);
JIG_STATUS_R_TRIG(CLK:= CONVEYOR.JIG_ST5.STATUS);
PROG_STEPS.ST5:=STEP;

END_PROGRAM

// ---- POUs/STATIONS/ST6_PMAX.TcPOU
PROGRAM ST6_PMAX
VAR
	STEP: INT := 0;
	JIG_STATUS_R_TRIG: R_TRIG;
	START_TAMPO_AMORCAGE: BOOL;
	TAMPO_AMORCAGE_TON: TON;
	START_TAMPO_MESURE: BOOL;
	TAMPO_MESURE_TON: TON;
	START_TAMPO_VIDANGE: BOOL;
	TAMPO_VIDANGE_TON: TON;
	TAMPO_SORTIE_VERIN_HAUT_TON: TON;
	START_TAMPO_VERIN_HAUT: BOOL;
	TAMPO_SORTIE_VERIN_BAS_TON: TON;
	START_TAMPO_VERIN_BAS: BOOL;
	TAMPO_SORTIE_VERIN_ELEC_TON: TON;
	START_TAMPO_VERIN_ELEC: BOOL;
	START_TAMPO_MESURE_PERTES: BOOL;
	TAMPO_MESURE_PERTES_TON: TON;
	TEMPS_VIDA: TIME;
END_VAR

(*******************************************************
*
* Station 6 - Pression MAX
*
*
*********************************************************)
IF NOT(GEMMA.STEP='F1') THEN
	STEP:=0;
END_IF;


CASE STEP OF

0: (*Init*)

	ST6_6V4 := FALSE;
	ST6_6V5 := FALSE;
	ST6_6V6 := FALSE;
	ST6_6V6 := FALSE;
	ST6_6V7 := FALSE;
	ST6_6V10 := FALSE;
	ST6_6V11 := FALSE;
	
	FLAGS.ST6_RELEASE_CARRIER := FALSE;
	START_TAMPO_AMORCAGE := FALSE;
	START_TAMPO_MESURE:= FALSE;
	START_TAMPO_MESURE_PERTES:= FALSE;
	START_TAMPO_VIDANGE:= FALSE;
	START_TAMPO_VERIN_ELEC := FALSE;
	START_TAMPO_VERIN_HAUT := FALSE;
	START_TAMPO_VERIN_BAS := FALSE;
	
	STEP := STEP + 10;
	
10: (*Attend une palette / flanc montant du status*)

	IF JIG_STATUS_R_TRIG.Q THEN
		STEP := STEP + 10;
	END_IF;
	
20: (*Descend le vérin du dessus*)

	ST6_6V4 := TRUE;
	START_TAMPO_VERIN_HAUT := TRUE;
	STEP := STEP + 10;
	
30: (*Attend vérin dessus sorti*)

	IF TAMPO_SORTIE_VERIN_HAUT_TON.Q THEN
		START_TAMPO_VERIN_HAUT := FALSE;
		STEP := STEP + 10;
	END_IF;

40: (*Monte le vérin du dessous*)

	ST6_6V5 := TRUE;
	START_TAMPO_VERIN_BAS := TRUE;
	STEP := STEP + 10;
	
50: (*Attend vérin dessus sorti*)

	IF TAMPO_SORTIE_VERIN_BAS_TON.Q THEN
		START_TAMPO_VERIN_BAS := FALSE;
		STEP := STEP + 10;
	END_IF;
	
60: (*Sort le vérin électrique*)

	ST6_6V6 := TRUE;
	IF PUMP_PARAMS.GEN_BYPASS THEN
		ST6_6V7 := TRUE;
	END_IF
	START_TAMPO_VERIN_ELEC := TRUE;
	STEP := STEP + 10;
	
70: (*Attend vérin électrique sortie*)

	IF TAMPO_SORTIE_VERIN_ELEC_TON.Q THEN
		START_TAMPO_VERIN_ELEC := FALSE;
		STEP := STEP + 10;
	END_IF;

80: (*Allume la pompe*)

	ST6_POWER := TRUE;
	ST6_6V10 := TRUE;
	ST6_6V11 := TRUE;
	STEP := 100;
	
	
(**************************************************************************)
100: (*Démarre la tampo pour l'amorcage*)

	START_TAMPO_AMORCAGE := TRUE;
	STEP := STEP + 10;
	
110: (*Attend fin tampo amorcage*)

	IF TAMPO_AMORCAGE_TON.Q THEN
		START_TAMPO_AMORCAGE := FALSE;
		STEP := STEP + 10;
	END_IF;
	
120: (*Démarre la tampo pour la mesure de pression*)

	START_TAMPO_MESURE := TRUE;
	ST6_6V11 := FALSE; 		(*ferme la vanne après la pompe *)
	STEP := STEP + 10;
	
130: (*Attend fin tampo mesure - MESURE EN COURT*)

	IF TAMPO_MESURE_TON.Q THEN
		START_TAMPO_MESURE := FALSE;
		ST6_6V11 := TRUE; 		(*re-ouvre la vanne après la pompe *)
		STEP := STEP + 10;
	END_IF;
	
140: (*Démarre la tampo pour la mesure de perte de pression*)

	START_TAMPO_MESURE_PERTES := TRUE;
	ST6_POWER := FALSE;
	STEP := STEP + 10;
	
150: (*Attend fin tampo mesure - MESURE EN COURT perte de pression*)

	IF TAMPO_MESURE_PERTES_TON.Q THEN
		START_TAMPO_MESURE_PERTES := FALSE;
		STEP := 300;
	END_IF;
	

(**************************************************************************)	

300: (*Descend le vérin du dessous*)

	ST6_6V5 := FALSE;
	ST6_6V10 := FALSE;	(* ferme la vanne avant la pompe*)
	STEP := STEP + 10;

310: (*Démarre la tampo de vidange de la pompe*)

	START_TAMPO_VIDANGE := TRUE;
	STEP := STEP + 10;
	
320: (*Attend fin tampo amorcage*)

	IF TAMPO_VIDANGE_TON.Q THEN
		START_TAMPO_VIDANGE := FALSE;
		ST6_6V11 := FALSE; (* ferme la vanne après la pompe*)
		STEP := STEP + 10;
	END_IF;

330: (*Rentre le vérin électrique*)

	ST6_6V6 := FALSE;
	ST6_6V7 := FALSE;
	STEP := STEP + 10;
	
	
340: (*Monte le vérin du dessus*)

	ST6_6V4 := FALSE;
	STEP := STEP + 10;

350: (*Libère la palette*)

	FLAGS.ST6_RELEASE_CARRIER := TRUE;
	STEP := 0;


ELSE
    (*default case*);
END_CASE;

(*FBs*)
TAMPO_SORTIE_VERIN_HAUT_TON(IN:= START_TAMPO_VERIN_HAUT, PT:= TEMPS_SORTIE_VERIN);
TAMPO_SORTIE_VERIN_BAS_TON(IN:= START_TAMPO_VERIN_BAS, PT:= TEMPS_SORTIE_VERIN);
TAMPO_SORTIE_VERIN_ELEC_TON(IN:= START_TAMPO_VERIN_ELEC, PT:= TEMPS_SORTIE_VERIN);

TAMPO_AMORCAGE_TON(IN:= START_TAMPO_AMORCAGE, PT:= PUMP_PARAMS.ST6_TEMPS_POMPAGE);
TAMPO_VIDANGE_TON(IN:= START_TAMPO_VIDANGE, PT:= TEMPS_VIDANGE_POMPE);
TAMPO_MESURE_TON(IN:= START_TAMPO_MESURE, PT:= PUMP_PARAMS.ST6_TEMPS_MESURE);
TAMPO_MESURE_PERTES_TON(IN:= START_TAMPO_MESURE_PERTES, PT:= PUMP_PARAMS.ST6_TEMPS_MESURE_PERTE_PRESSION);
JIG_STATUS_R_TRIG(CLK:= CONVEYOR.JIG_ST6.STATUS);
PROG_STEPS.ST6:=STEP;

END_PROGRAM

// ---- POUs/STATIONS/ST7_SECHAGE.TcPOU
PROGRAM ST7_SECHAGE
VAR
	STEP: INT := 0;
	START_TAMPO_AIR: BOOL;
	TAMPO_AIR: TON;
	JIG_STATUS_R_TRIG: R_TRIG;
	TAMPO_SORTIE_VERIN_HAUT_TON: TON;
	START_TAMPO_VERIN_HAUT: BOOL;
	TAMPO_SORTIE_VERIN_BAS_TON: TON;
	START_TAMPO_VERIN_BAS: BOOL;
	TAMPO_SORTIE_VERIN_ELEC_TON: TON;
	START_TAMPO_VERIN_ELEC: BOOL;
END_VAR

(*******************************************************
*
* Station 7 - Séchage
*
*
*********************************************************)
IF NOT(GEMMA.STEP='F1') THEN
	STEP:=0;
END_IF;


CASE STEP OF

0: (*Init*)

	ST7_7V4 := FALSE;
	ST7_7V5 := FALSE;
	ST7_7V6 := FALSE;
	ST7_7V7 := FALSE;
	
	FLAGS.ST7_RELEASE_CARRIER := FALSE;
	START_TAMPO_AIR := FALSE;
	
	STEP := STEP + 10;
	
10: (*Attend une palette / flanc montant du status*)

	IF JIG_STATUS_R_TRIG.Q THEN
		STEP := STEP + 10;
	END_IF;
	
20: (*Descend le vérin du dessus*)

	ST7_7V4 := TRUE;
	STEP := STEP + 10;
	START_TAMPO_VERIN_HAUT:=TRUE;
	
30: (*Attend vérin dessus sorti*)

	IF TAMPO_SORTIE_VERIN_HAUT_TON.Q THEN
		START_TAMPO_VERIN_HAUT := FALSE;
		STEP := STEP + 10;
	END_IF;

40: (*Monte le vérin du dessous*)

	ST7_7V5 := TRUE;
	START_TAMPO_VERIN_BAS:=TRUE;
	STEP := STEP + 10;
	
50: (*Attend vérin dessous sorti*)

	IF TAMPO_SORTIE_VERIN_BAS_TON.Q THEN
		START_TAMPO_VERIN_BAS:=FALSE;
		STEP := STEP + 10;
	END_IF;
	
60: (*Sort le vérin électrique*)

	ST7_7V6 := TRUE;
	IF PUMP_PARAMS.GEN_BYPASS THEN
		ST7_7V7 := TRUE;
	END_IF
	START_TAMPO_VERIN_ELEC:=TRUE;
	STEP := STEP + 10;
	
70: (*Attend vérin électrique sortie*)

	IF TAMPO_SORTIE_VERIN_ELEC_TON.Q THEN
		START_TAMPO_VERIN_ELEC:=FALSE;
		STEP := STEP + 10;
	END_IF;

80: (*Allume la pompe*)

	ST7_POWER := TRUE;
	STEP := 100;
	
(**************************************************************************)
100: (*ouvre l'air pour le séchage et démarre la tampo*)

	ST7_7V10 := TRUE;
	START_TAMPO_AIR :=TRUE;
	STEP := STEP + 10;
	
110: (*Attend fin tampo AIR et stop l'air*)

	IF TAMPO_AIR.Q THEN
		START_TAMPO_AIR := FALSE;
		ST7_7V10 := FALSE;
		STEP := 300;
	END_IF;

(**************************************************************************)	

300: (*Rentre le vérin électrique*)

	ST7_7V6 := FALSE;
	ST7_7V7 := FALSE;
	STEP := STEP + 10;
	
310: (*Descend le vérin du dessous*)

	ST7_7V5 := FALSE;
	STEP := STEP + 10;
	
320: (*Monte le vérin du dessus*)

	ST7_7V4 := FALSE;
	STEP := STEP + 10;

330: (*Libère la palette*)

	FLAGS.ST7_RELEASE_CARRIER := TRUE;
	STEP := 0;


ELSE
    (*default case*);
END_CASE;

(*FBs*)
TAMPO_SORTIE_VERIN_HAUT_TON(IN:= START_TAMPO_VERIN_HAUT, PT:= TEMPS_SORTIE_VERIN);
TAMPO_SORTIE_VERIN_BAS_TON(IN:= START_TAMPO_VERIN_BAS, PT:= TEMPS_SORTIE_VERIN);
TAMPO_SORTIE_VERIN_ELEC_TON(IN:= START_TAMPO_VERIN_ELEC, PT:= TEMPS_SORTIE_VERIN);
TAMPO_AIR(IN:= START_TAMPO_AIR, PT:= PUMP_PARAMS.ST7_TEMPS_SECHAGE);
JIG_STATUS_R_TRIG(CLK:= CONVEYOR.JIG_ST7.STATUS);
PROG_STEPS.ST7:=STEP;

END_PROGRAM

// ---- POUs/STATIONS/ST8_IMPRESSION.TcPOU
PROGRAM ST8_IMPRESSION
VAR
	STEP: INT := 0;
	JIG_STATUS_R_TRIG: R_TRIG;
END_VAR

(*******************************************************
*
* Station 8 - Impression
*
*
*********************************************************)
IF NOT(GEMMA.STEP='F1') THEN
	STEP:=0;
END_IF;


CASE STEP OF

0: (*Init*)
	
	ST8_PRET_A_IMPRIMER := FALSE;
	FLAGS.ST8_RELEASE_CARRIER := FALSE;
	
	STEP := STEP + 10;
	
10: (*Attend une palette / flanc montant du status*)

	IF JIG_STATUS_R_TRIG.Q THEN
		STEP := 100;
	END_IF;

	
(**************************************************************************)
100: (*Pompre prête*)
	
	ST8_PRET_A_IMPRIMER := TRUE;
	STEP := STEP + 10;
	
110: (*Attend fin de l'impression de l'étiquette*)

	IF ST8_IMPRESSION_OK THEN
		ST8_PRET_A_IMPRIMER := FALSE;
		STEP := 300;
	END_IF;
	

(**************************************************************************)	


300: (*Libère la palette*)

	FLAGS.ST8_RELEASE_CARRIER := TRUE;
	STEP := 0;


ELSE
    (*default case*);
END_CASE;

(*FBs*)
JIG_STATUS_R_TRIG(CLK:= CONVEYOR.JIG_ST8.STATUS);
PROG_STEPS.ST8:=STEP;

END_PROGRAM

// ---- POUs/STATIONS/ST9_DECHARGEMENT.TcPOU
PROGRAM ST9_DECHARGEMENT
VAR
	STEP: INT := 0;
	JIG_STATUS_R_TRIG: R_TRIG;
END_VAR

(*******************************************************
*
* Station 7 - Séchage
*
*
*********************************************************)
IF NOT(GEMMA.STEP='F1') THEN
	STEP:=0;
END_IF;


CASE STEP OF

0: (*Init*)

	ST9_9V4A := TRUE;
	ST9_9V4B := FALSE;
	ST9_9V5A := FALSE;
	ST9_9V5B := TRUE;
	ST9_9V6 := TRUE;
	ST9_9V7 := FALSE;
	
	FLAGS.ST9_RELEASE_CARRIER := FALSE;
	
	STEP := STEP + 10;
	
10: (*Attend une palette / flanc montant du status*)

	IF JIG_STATUS_R_TRIG.Q THEN
		IF ST9_DECHARGE THEN
			STEP := STEP + 10;
		ELSE
			STEP := 120;
		END_IF;
	END_IF;
	
20: (*Descend le vérin*)

	ST9_9V5A := TRUE;
	ST9_9V5B := FALSE;
	IF PUMP_PARAMS.ST9_BOBINE_A_FIL THEN
		ST9_9V7 := TRUE;
	END_IF;
	STEP := STEP + 10;
	
30: (*Attend que le vérin soit en bas*)

	IF ST9_9B51 THEN
		STEP := STEP + 10;
	END_IF;
	
40: (*Ferme la pince*)

	ST9_9V6 := FALSE;
	STEP := STEP + 10;
	
50: (*Attend que la pince soit fermée*)

	IF ST9_9B6 THEN
		STEP := STEP + 10;
	END_IF;
	
60: (*Monte*)

	ST9_9V5A := FALSE;
	ST9_9V5B := TRUE;
	STEP := STEP + 10;
	
70: (*Attend que le vérin soit en haut*)

	IF ST9_9B5 THEN
		FLAGS.ST9_RELEASE_CARRIER := TRUE;
		ST9_9V7 := FALSE;
		STEP := STEP + 10;
	END_IF;
	
80: (*Déplacement vers déchargement*)

	ST9_9V4A := FALSE;
	ST9_9V4B := TRUE;
	STEP := STEP + 10;
	
90: (*Attend que le vérin soit en haut*)

	IF ST9_9B4 THEN
		STEP := STEP + 10;
	END_IF;
	
100: (*Déplacement vers le bas*)

	ST9_9V5A := TRUE;
	ST9_9V5B := FALSE;
	STEP := STEP + 10;
	
110: (*Attend que le vérin soit en haut*)

	IF ST9_9B51 THEN
		STEP := STEP + 10;
	END_IF;
	
120: (*Libère la pompe*)
	
	ST9_9V6 := TRUE;
	STEP := STEP + 10;
	
130: (*Attend libération*)

	IF ST9_9B6 THEN
		STEP := STEP + 10;
	END_IF;

140: (*Monte*)

	ST9_9V5A := FALSE;
	ST9_9V5B := TRUE;
	STEP := STEP + 10;
	
150: (*Attend vérin en haut*)

	IF ST9_9B5 THEN
		STEP := STEP + 10;
	END_IF;
	
160: (*Retour vers palette*)

	ST9_9V4A := TRUE;
	ST9_9V4B := FALSE;
	STEP := STEP + 10;
	
170: (*Attend vérin en haut*)

	IF ST9_9B41 THEN
		FLAGS.ST9_RELEASE_CARRIER := TRUE;
		STEP := 0;
	END_IF;



ELSE
    (*default case*);
END_CASE;

(*FBs*)

JIG_STATUS_R_TRIG(CLK:= CONVEYOR.JIG_ST9.STATUS);
PROG_STEPS.ST9:=STEP;

END_PROGRAM

// ---- POUs/Functions/PRESSURE_REGULATOR.TcPOU
FUNCTION_BLOCK PRESSURE_REGULATOR
VAR_INPUT
	COURANT			: LREAL;
	PRESSION_CONSIGNE : REAL;
	PRESSION_MESURE : REAL;
	MOTOR_POSITION_MAX :FLOAT;
	MOTOR_INITIAL_POSITION: LREAL;
	GEMMA	:STRING;
END_VAR
VAR_OUTPUT
	MOTOR_POSITION 	: DINT;
END_VAR
VAR
	gainScheduled_Kp			: REAL;
	gainScheduled_Ki			: REAL;
	gainScheduled_Kd			: REAL;
	P_ERREUR:REAL;
	GAIN:REAL:=4.0;
	

	eMode						: E_CTRL_MODE;
	stCTRL_PID_PARAMS			: ST_CTRL_PID_PARAMS;

	eErrorId					: E_CTRL_ERRORCODES;
	bError						: BOOL;
	bARWactive					: BOOL;

	(* controller  *)
	fbCTRL_PID					: FB_CTRL_PID;

	fOut: LREAL;
	bHold: BOOL;
END_VAR

IF PUMP_PARAMS.GEN_GRAND_DEBIT=FALSE THEN (*USING STATION 4*)
	IF PRESSION_CONSIGNE>ST4_PID_HighPressure.q THEN
		(*Utilise le régulateur pour les hautes pression*)
		gainScheduled_Kp:=ST4_PID_HighPressure.Kp;
		gainScheduled_Ki:=ST4_PID_HighPressure.Ki;
		gainScheduled_Kd:=ST4_PID_HighPressure.Kd;
	ELSIF PRESSION_CONSIGNE<=ST4_PID_HighPressure.q AND PRESSION_CONSIGNE>ST4_PID_MiddlePressure.q THEN
		(*Calcule les paramètres du régulateur avec une interpolation linéaire entre un PID prévu pour les hautes pressions et un PID pour les moyennes pressions*)
		gainScheduled_Kp:=(ST4_PID_HighPressure.q-PRESSION_CONSIGNE)/(ST4_PID_HighPressure.q-ST4_PID_MiddlePressure.q)*ST4_PID_MiddlePressure.Kp+(PRESSION_CONSIGNE-ST4_PID_MiddlePressure.q)/(ST4_PID_HighPressure.q-ST4_PID_MiddlePressure.q)*ST4_PID_HighPressure.Kp;
		gainScheduled_Ki:=(ST4_PID_HighPressure.q-PRESSION_CONSIGNE)/(ST4_PID_HighPressure.q-ST4_PID_MiddlePressure.q)*ST4_PID_MiddlePressure.Ki+(PRESSION_CONSIGNE-ST4_PID_MiddlePressure.q)/(ST4_PID_HighPressure.q-ST4_PID_MiddlePressure.q)*ST4_PID_HighPressure.Ki;
		gainScheduled_Kd:=(ST4_PID_HighPressure.q-PRESSION_CONSIGNE)/(ST4_PID_HighPressure.q-ST4_PID_MiddlePressure.q)*ST4_PID_MiddlePressure.Kd+(PRESSION_CONSIGNE-ST4_PID_MiddlePressure.q)/(ST4_PID_HighPressure.q-ST4_PID_MiddlePressure.q)*ST4_PID_HighPressure.Kd;
	ELSIF PRESSION_CONSIGNE<=ST4_PID_MiddlePressure.q AND PRESSION_CONSIGNE>ST4_PID_LowPressure.q THEN
		(*Calcule les paramètres du régulateur avec une interpolation linéaire entre un PID prévu pour les moyennes pressions et un PID pour les basses pressions*)
		gainScheduled_Kp:=(ST4_PID_MiddlePressure.q-PRESSION_CONSIGNE)/(ST4_PID_MiddlePressure.q-ST4_PID_LowPressure.q)*ST4_PID_LowPressure.Kp+(PRESSION_CONSIGNE-ST4_PID_LowPressure.q)/(ST4_PID_MiddlePressure.q-ST4_PID_LowPressure.q)*ST4_PID_MiddlePressure.Kp;
		gainScheduled_Ki:=(ST4_PID_MiddlePressure.q-PRESSION_CONSIGNE)/(ST4_PID_MiddlePressure.q-ST4_PID_LowPressure.q)*ST4_PID_LowPressure.Ki+(PRESSION_CONSIGNE-ST4_PID_LowPressure.q)/(ST4_PID_MiddlePressure.q-ST4_PID_LowPressure.q)*ST4_PID_MiddlePressure.Ki;
		gainScheduled_Kd:=(ST4_PID_MiddlePressure.q-PRESSION_CONSIGNE)/(ST4_PID_MiddlePressure.q-ST4_PID_LowPressure.q)*ST4_PID_LowPressure.Kd+(PRESSION_CONSIGNE-ST4_PID_LowPressure.q)/(ST4_PID_MiddlePressure.q-ST4_PID_LowPressure.q)*ST4_PID_MiddlePressure.Kd;
	ELSE (*PRESSION_CONSIGNE<ST4_PID_LowPressure.q*)
		(*Utilise le régulateur pour les basses pressions*)
		gainScheduled_Kp:=ST4_PID_LowPressure.Kp;
		gainScheduled_Ki:=ST4_PID_LowPressure.Ki;
		gainScheduled_Kd:=ST4_PID_LowPressure.Kd;	
	END_IF 
ELSE (*USING STATION 5*)
	(*Utilise le régulateur pour les pressions moyennes*)
	IF PRESSION_CONSIGNE>ST5_PID_MiddlePressure.q THEN
		gainScheduled_Kp:=ST5_PID_MiddlePressure.Kp;
		gainScheduled_Ki:=ST5_PID_MiddlePressure.Ki;
		gainScheduled_Kd:=ST5_PID_MiddlePressure.Kd;	
	ELSIF PRESSION_CONSIGNE<=ST5_PID_MiddlePressure.q AND PRESSION_CONSIGNE>ST5_PID_LowPressure.q THEN
		(*Calcule les paramètres du régulateur avec une interpolation linéaire entre un PID prévu pour les moyennes pressions et un PID pour les basses pressions*)
		gainScheduled_Kp:=(ST5_PID_MiddlePressure.q-PRESSION_CONSIGNE)/(ST5_PID_MiddlePressure.q-ST5_PID_LowPressure.q)*ST5_PID_LowPressure.Kp+(PRESSION_CONSIGNE-ST5_PID_LowPressure.q)/(ST5_PID_MiddlePressure.q-ST5_PID_LowPressure.q)*ST5_PID_MiddlePressure.Kp;
		gainScheduled_Ki:=(ST5_PID_MiddlePressure.q-PRESSION_CONSIGNE)/(ST5_PID_MiddlePressure.q-ST5_PID_LowPressure.q)*ST5_PID_LowPressure.Ki+(PRESSION_CONSIGNE-ST5_PID_LowPressure.q)/(ST5_PID_MiddlePressure.q-ST5_PID_LowPressure.q)*ST5_PID_MiddlePressure.Ki;
		gainScheduled_Kd:=(ST5_PID_MiddlePressure.q-PRESSION_CONSIGNE)/(ST5_PID_MiddlePressure.q-ST5_PID_LowPressure.q)*ST5_PID_LowPressure.Kd+(PRESSION_CONSIGNE-ST5_PID_LowPressure.q)/(ST5_PID_MiddlePressure.q-ST5_PID_LowPressure.q)*ST5_PID_MiddlePressure.Kd;
	ELSE (*PRESSION_CONSIGNE<ST5_PID_LowPressure.q*)
		(*Utilise le régulateur pour les basses pressions*)
		gainScheduled_Kp:=ST5_PID_LowPressure.Kp;
		gainScheduled_Ki:=ST5_PID_LowPressure.Ki;
		gainScheduled_Kd:=ST5_PID_LowPressure.Kd;
	END_IF
END_IF

	(* init parameter struct *)
	stCTRL_PID_PARAMS.tCtrlCycleTime		:= T#10MS;
	stCTRL_PID_PARAMS.tTaskCycleTime		:= T#10MS;
	stCTRL_PID_PARAMS.tTn					:= REAL_TO_TIME(gainScheduled_Ki);			(* integral gain tTn				*)
	stCTRL_PID_PARAMS.tTv					:= REAL_TO_TIME(gainScheduled_Kd);			(* derivative gain tTv				*)
	stCTRL_PID_PARAMS.tTd					:= stCTRL_PID_PARAMS.tTv/5;					(* filter parameter for the real derivative gain part *)
	stCTRL_PID_PARAMS.fKp					:= gainScheduled_Kp;						(* proportional gain Kp				*)
	stCTRL_PID_PARAMS.fOutMaxLimit			:= MOTOR_POSITION_MAX;		  				(* maximum output limit				*)
	stCTRL_PID_PARAMS.fOutMinLimit			:= 0;										(* minimum output limit				*)
	stCTRL_PID_PARAMS.bPInTheFeedbackPath 	:= FALSE;									(* let it to false for a standart PID transfert function *)
    stCTRL_PID_PARAMS.bDInTheFeedbackPath 	:= FALSE;
    stCTRL_PID_PARAMS.bARWOnIPartOnly   	:= TRUE;									(* anti-reset windup *)
	(* set the mode to ACTIVE --> normal operation *)
	eMode							:= eCTRL_MODE_ACTIVE;

	(*Fixe la valeur d'entrée initiale pour le moteur en A1*)
	IF GEMMA = 'A1' THEN
		bHold :=TRUE;
	ELSE
		bHold :=FALSE;
	END_IF

	(*Controller pour la pression*)
	fbCTRL_PID(		fSetpointValue		:= PRESSION_CONSIGNE,
					fActualValue		:= PRESSION_MESURE,
					fManSyncValue		:= MOTOR_INITIAL_POSITION,
					bSync				:= bHold,
					eMode				:= eMode,
					bHold				:= bHold,
					stParams			:= stCTRL_PID_PARAMS,
					fOut				=> fOut,
					bARWactive			=> bARWactive,
					eErrorId			=> eErrorId,
					bError				=> bError
	);
	
MOTOR_POSITION := LREAL_TO_DINT(fOut);



(*	
P_ERREUR:=PRESSION_CONSIGNE - PRESSION_MESURE;

IF COURANT > 10.0 THEN
	MOTOR_POSITION := MOTOR_POSITION + REAL_TO_INT(P_ERREUR*GAIN);(* P_ERREUR*GAIN *)
END_IF;*)

END_FUNCTION_BLOCK

// ---- POUs/EH/EH_FLOMETER.TcPOU
FUNCTION_BLOCK EH_FLOMETER

VAR_INPUT
	AI1: ARRAY [0..4] OF USINT;
	AI2: ARRAY [0..4] OF USINT;
	AI3: ARRAY [0..4] OF USINT;
	AI4: ARRAY [0..4] OF USINT;
	AI5: ARRAY [0..4] OF USINT;
	AI6: ARRAY [0..4] OF USINT;
	TOT: ARRAY [0..4] OF USINT;
END_VAR

VAR_OUTPUT
	MassFlow: REAL;
	VolumeFlow: REAL;
	CorrectedVolueFLow: REAL;
	Density: REAL;
	ReferenceDensity:REAL;
	Temperature:REAL;
	TotalMass: REAL;
END_VAR

VAR

END_VAR

MassFlow:=EH_IEEE754_TO_REAL(AI1);
VolumeFlow:=EH_IEEE754_TO_REAL(AI2);
CorrectedVolueFLow:=EH_IEEE754_TO_REAL(AI3);
Density:=EH_IEEE754_TO_REAL(AI4);
ReferenceDensity:=EH_IEEE754_TO_REAL(AI5);
Temperature:=EH_IEEE754_TO_REAL(AI6);
TotalMass:=EH_IEEE754_TO_REAL(TOT);

END_FUNCTION_BLOCK

// ---- POUs/EH/EH_IEEE754_TO_REAL.TcPOU
FUNCTION EH_IEEE754_TO_REAL : REAL
VAR_INPUT
	AI: ARRAY [0..4] OF USINT;
END_VAR

VAR
	Sign: SINT;
	Exponent:INT;
	Mantisse: REAL;
END_VAR

Sign:=		BOOL_TO_SINT(AI[0].7)*-1;

Exponent:= 	BOOL_TO_SINT(AI[1].7)*1 +
			BOOL_TO_SINT(AI[0].0)*2 +
			BOOL_TO_SINT(AI[0].1)*4 +
			BOOL_TO_SINT(AI[0].2)*8 +
			BOOL_TO_SINT(AI[0].3)*16 +
			BOOL_TO_SINT(AI[0].4)*32 +
			BOOL_TO_SINT(AI[0].5)*64 +
			BOOL_TO_SINT(AI[0].6)*128;

(*met à zéro le bit 7 du byte 1 qui n'est pas dans le mantisse*)
AI[1].7:=0;

Mantisse:=	BOOL_TO_SINT(AI[1].0)*EXPT(2,-7) +
			BOOL_TO_SINT(AI[1].1)*EXPT(2,-6) +
			BOOL_TO_SINT(AI[1].2)*EXPT(2,-5) +
			BOOL_TO_SINT(AI[1].3)*EXPT(2,-4) +
			BOOL_TO_SINT(AI[1].4)*EXPT(2,-3) +
			BOOL_TO_SINT(AI[1].5)*EXPT(2,-2) +
			BOOL_TO_SINT(AI[1].6)*EXPT(2,-1) +
			BOOL_TO_SINT(AI[2].0)*EXPT(2,-15) +
			BOOL_TO_SINT(AI[2].1)*EXPT(2,-14) +
			BOOL_TO_SINT(AI[2].2)*EXPT(2,-13) +
			BOOL_TO_SINT(AI[2].3)*EXPT(2,-12) +
			BOOL_TO_SINT(AI[2].4)*EXPT(2,-11) +
			BOOL_TO_SINT(AI[2].5)*EXPT(2,-10) +
			BOOL_TO_SINT(AI[2].6)*EXPT(2,-9) +
			BOOL_TO_SINT(AI[2].7)*EXPT(2,-8) +
			BOOL_TO_SINT(AI[3].0)*EXPT(2,-23) +
			BOOL_TO_SINT(AI[3].1)*EXPT(2,-22) +
			BOOL_TO_SINT(AI[3].2)*EXPT(2,-21) +
			BOOL_TO_SINT(AI[3].3)*EXPT(2,-20) +
			BOOL_TO_SINT(AI[3].4)*EXPT(2,-19) +
			BOOL_TO_SINT(AI[3].5)*EXPT(2,-18) +
			BOOL_TO_SINT(AI[3].6)*EXPT(2,-17) +
			BOOL_TO_SINT(AI[3].7)*EXPT(2,-16);

EH_IEEE754_TO_REAL:=EXPT(-1,Sign)*EXPT(2,Exponent-127)*(1+Mantisse);

IF EH_IEEE754_TO_REAL<0.000001 THEN
EH_IEEE754_TO_REAL:=0;
END_IF;

END_FUNCTION

// ---- POUs/MAXON/ST5_MOTOR_1.TcPOU
PROGRAM ST5_MOTOR_1
VAR
	ClearFault: FB_ClearFault;
	SetEnableState: FB_SetEnableState;
	SetHomingParameter: FB_SetHomingParameter;
	FindHome: FB_FindHome;
	POSITION: DINT;
	GetMovementState: FB_GetMovementState;
	MoveToPosition: FB_MoveToPosition;
	SetOperationMode: FB_SetOperationMode;
	SetMotorParameter: FB_SetMotorParameter;
	SetPositionProfile: FB_SetPositionProfile;
END_VAR

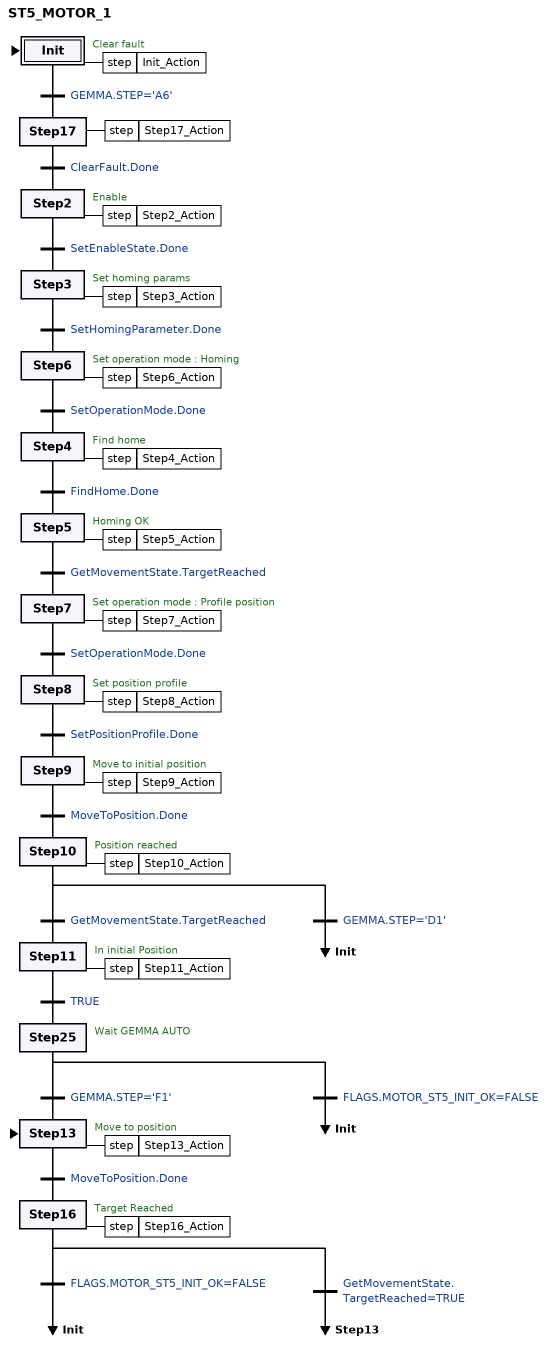
// Clear fault
INITIAL_STEP Init:
    Init_Action(N);  // step action
END_STEP
TRANSITION FROM Init TO Step17
    := GEMMA.STEP='A6';
END_TRANSITION
STEP Step17:
    Step17_Action(N);  // step action
END_STEP
TRANSITION FROM Step17 TO Step2
    := ClearFault.Done;
END_TRANSITION
// Enable
STEP Step2:
    Step2_Action(N);  // step action
END_STEP
TRANSITION FROM Step2 TO Step3
    := SetEnableState.Done;
END_TRANSITION
// Set homing params
STEP Step3:
    Step3_Action(N);  // step action
END_STEP
TRANSITION FROM Step3 TO Step6
    := SetHomingParameter.Done;
END_TRANSITION
// Set operation mode : Homing
STEP Step6:
    Step6_Action(N);  // step action
END_STEP
TRANSITION FROM Step6 TO Step4
    := SetOperationMode.Done;
END_TRANSITION
// Find home
STEP Step4:
    Step4_Action(N);  // step action
END_STEP
TRANSITION FROM Step4 TO Step5
    := FindHome.Done;
END_TRANSITION
// Homing OK
STEP Step5:
    Step5_Action(N);  // step action
END_STEP
TRANSITION FROM Step5 TO Step7
    := GetMovementState.TargetReached;
END_TRANSITION
// Set operation mode : Profile position
STEP Step7:
    Step7_Action(N);  // step action
END_STEP
TRANSITION FROM Step7 TO Step8
    := SetOperationMode.Done;
END_TRANSITION
// Set position profile
STEP Step8:
    Step8_Action(N);  // step action
END_STEP
TRANSITION FROM Step8 TO Step9
    := SetPositionProfile.Done;
END_TRANSITION
// Move to initial position
STEP Step9:
    Step9_Action(N);  // step action
END_STEP
TRANSITION FROM Step9 TO Step10
    := MoveToPosition.Done;
END_TRANSITION
// Position reached
STEP Step10:
    Step10_Action(N);  // step action
END_STEP
TRANSITION FROM Step10 TO Step11
    := GetMovementState.TargetReached;
END_TRANSITION
TRANSITION FROM Step10 TO Init
    := GEMMA.STEP='D1';
END_TRANSITION
// In initial Position
STEP Step11:
    Step11_Action(N);  // step action
END_STEP
TRANSITION FROM Step11 TO Step25
    := TRUE;
END_TRANSITION
// Wait GEMMA AUTO
STEP Step25:
END_STEP
TRANSITION FROM Step25 TO Step13
    := GEMMA.STEP='F1';
END_TRANSITION
TRANSITION FROM Step25 TO Init
    := FLAGS.MOTOR_ST5_INIT_OK=FALSE;
END_TRANSITION
// Move to position
STEP Step13:
    Step13_Action(N);  // step action
END_STEP
TRANSITION FROM Step13 TO Step16
    := MoveToPosition.Done;
END_TRANSITION
// Target Reached
STEP Step16:
    Step16_Action(N);  // step action
END_STEP
TRANSITION FROM Step16 TO Init
    := FLAGS.MOTOR_ST5_INIT_OK=FALSE;
END_TRANSITION
TRANSITION FROM Step16 TO Step13
    := GetMovementState.TargetReached=TRUE;
END_TRANSITION

ACTION Step6_Action:
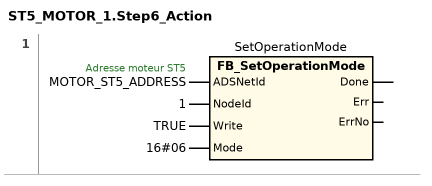
// NETWORK 1
//   MOTOR_ST5_ADDRESS: Adresse moteur ST5
SetOperationMode(ADSNetId := MOTOR_ST5_ADDRESS, NodeId := 1, Write := TRUE, Mode := 16#06); // FB_SetOperationMode
END_ACTION

ACTION Step2_Action:
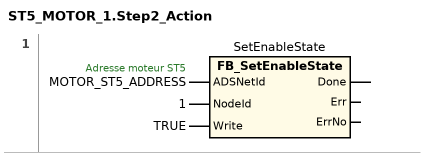
// NETWORK 1
//   MOTOR_ST5_ADDRESS: Adresse moteur ST5
SetEnableState(ADSNetId := MOTOR_ST5_ADDRESS, NodeId := 1, Write := TRUE); // FB_SetEnableState
END_ACTION

ACTION Step10_Action:
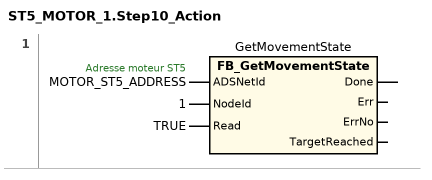
// NETWORK 1
//   MOTOR_ST5_ADDRESS: Adresse moteur ST5
GetMovementState(ADSNetId := MOTOR_ST5_ADDRESS, NodeId := 1, Read := TRUE); // FB_GetMovementState
END_ACTION

ACTION Step8_Action:
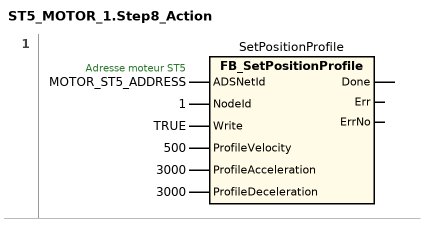
// NETWORK 1
//   MOTOR_ST5_ADDRESS: Adresse moteur ST5
SetPositionProfile(
    ADSNetId := MOTOR_ST5_ADDRESS,
    NodeId := 1,
    Write := TRUE,
    ProfileVelocity := 500,
    ProfileAcceleration := 3000,
    ProfileDeceleration := 3000); // FB_SetPositionProfile
END_ACTION

ACTION Step4_Action:
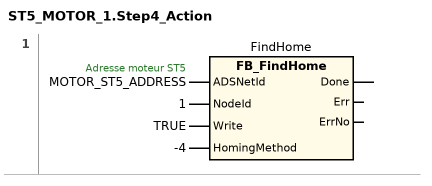
// NETWORK 1
//   MOTOR_ST5_ADDRESS: Adresse moteur ST5
FindHome(ADSNetId := MOTOR_ST5_ADDRESS, NodeId := 1, Write := TRUE, HomingMethod := -4); // FB_FindHome
END_ACTION

ACTION Step11_Action:

(*SetDisableState(
	ADSNetId:= '10.0.0.31.6.1',
	NodeId:= 1,
	Write:= TRUE);*)

FLAGS.MOTOR_ST5_INIT_OK:=TRUE;
END_ACTION

ACTION Step17_Action:
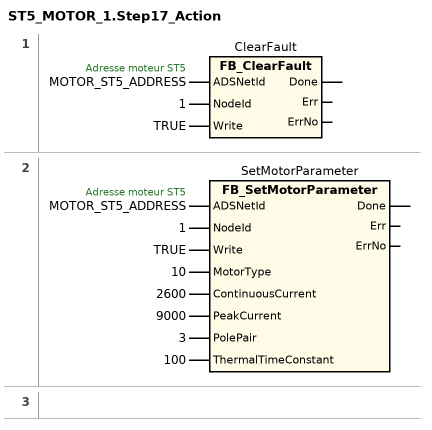
// NETWORK 1
//   MOTOR_ST5_ADDRESS: Adresse moteur ST5
ClearFault(ADSNetId := MOTOR_ST5_ADDRESS, NodeId := 1, Write := TRUE); // FB_ClearFault

// NETWORK 2
//   MOTOR_ST5_ADDRESS: Adresse moteur ST5
SetMotorParameter(
    ADSNetId := MOTOR_ST5_ADDRESS,
    NodeId := 1,
    Write := TRUE,
    MotorType := 10,
    ContinuousCurrent := 2600,
    PeakCurrent := 9000,
    PolePair := 3,
    ThermalTimeConstant := 100); // FB_SetMotorParameter

// NETWORK 3
END_ACTION

ACTION Step5_Action:
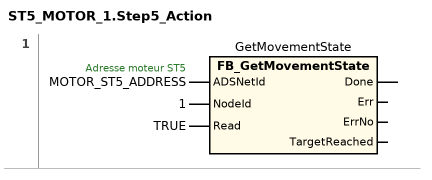
// NETWORK 1
//   MOTOR_ST5_ADDRESS: Adresse moteur ST5
GetMovementState(ADSNetId := MOTOR_ST5_ADDRESS, NodeId := 1, Read := TRUE); // FB_GetMovementState
END_ACTION

ACTION Step16_Action:
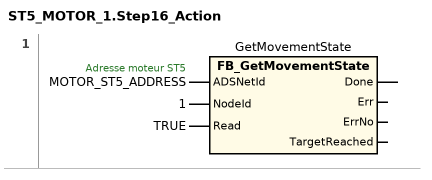
// NETWORK 1
//   MOTOR_ST5_ADDRESS: Adresse moteur ST5
GetMovementState(ADSNetId := MOTOR_ST5_ADDRESS, NodeId := 1, Read := TRUE); // FB_GetMovementState
END_ACTION

ACTION Init_Action:

END_ACTION

ACTION Step13_Action:
(*Limitation deplacement Moteur*)
IF FLAGS.MOTOR_ST5_POSITION>MOTOR_ST5_POSITION_MAX THEN
	POSITION:=MOTOR_ST5_POSITION_MAX;
ELSIF FLAGS.MOTOR_ST5_POSITION<0 THEN
	POSITION:=0;
ELSE
	POSITION:=FLAGS.MOTOR_ST5_POSITION;
END_IF


MoveToPosition(
	ADSNetId:= MOTOR_ST5_ADDRESS,
	NodeId:= 1,
	Write:= TRUE,
	TargetPosition:= POSITION,
	Absolut:= TRUE);
END_ACTION

ACTION Step3_Action:
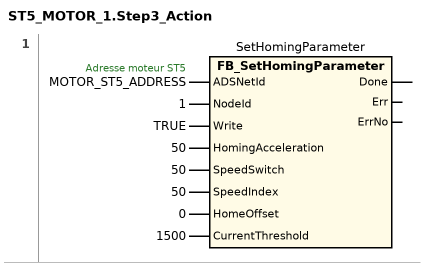
// NETWORK 1
//   MOTOR_ST5_ADDRESS: Adresse moteur ST5
SetHomingParameter(
    ADSNetId := MOTOR_ST5_ADDRESS,
    NodeId := 1,
    Write := TRUE,
    HomingAcceleration := 50,
    SpeedSwitch := 50,
    SpeedIndex := 50,
    HomeOffset := 0,
    CurrentThreshold := 1500); // FB_SetHomingParameter
END_ACTION

ACTION Step7_Action:
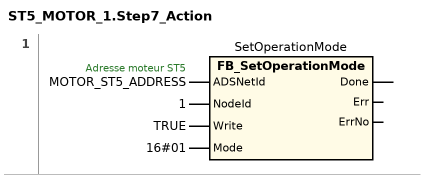
// NETWORK 1
//   MOTOR_ST5_ADDRESS: Adresse moteur ST5
SetOperationMode(ADSNetId := MOTOR_ST5_ADDRESS, NodeId := 1, Write := TRUE, Mode := 16#01); // FB_SetOperationMode
END_ACTION

ACTION Step9_Action:
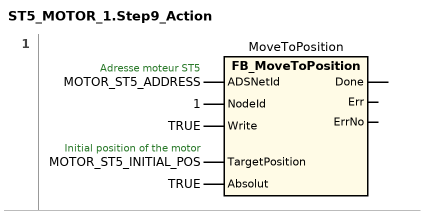
// NETWORK 1
//   MOTOR_ST5_ADDRESS: Adresse moteur ST5
//   MOTOR_ST5_INITIAL_POS: Initial position of the motor
MoveToPosition(
    ADSNetId := MOTOR_ST5_ADDRESS,
    NodeId := 1,
    Write := TRUE,
    TargetPosition := MOTOR_ST5_INITIAL_POS,
    Absolut := TRUE); // FB_MoveToPosition
END_ACTION

END_PROGRAM

// ---- POUs/STATIONS/Q1.TcPOU
PROGRAM Q1
VAR
	STEP: INT := 0;
	R_TRIG1:R_TRIG;
	FlowStop_Delay: TON;
	Start_FlowStop_Delay: BOOL;
	Pump_Delay: TON;
	Start_Pump_Delay: BOOL;
	Start_Suction_Delay: BOOL;
	Measurement_Delay: TON;
	Start_Measurement_Delay: BOOL;
	Init_Mass:REAL;

	FB_FormatString1: FB_FormatString;
	sInsertString: STRING;
	bError: BOOL;
	nErrid: DWORD;
	bBusyInsert: BOOL;
	bErrInsert: BOOL;
	nErridInsert: DWORD;
	FB_FormatStringDateTime: FB_FormatString;
	NT_GetTime1: NT_GetTime;
	tTime: TIMESTRUCT;
	bTimestart: BOOL:=0;
	sDateTimeString: T_MaxString;
	bExec_DBRecordInsert1: BOOL;
	P_ERREUR: REAL;
END_VAR

(*******************************************************
*
* Program fro the Q1 Test station
*
*
*********************************************************)
IF GEMMA.STEP='A6' THEN
	STEP:=0;
END_IF;


CASE STEP OF

0: (*Init*)
	Start_Pump_Delay:=FALSE;
	Start_FlowStop_Delay:=FALSE;
	Start_Measurement_Delay:=FALSE;
	Q1_DO.MAX_FLOW_VALVE:=FALSE;
	FLAGS.Q1_STATUS:=0;
	FLAGS.Q1_RELEASE_CARRIER:=0;
	Q1_FLOWMETER_CONTROL.SET_TOT:=1; (*Reset mass flow counter*)
	STEP := STEP+10;

10: (*Wait main JIG Ready*)
	IF R_TRIG1.Q AND GEMMA.STEP='F1'  THEN
		FLAGS.Q1_STATUS:=1;
		Q1_FLOWMETER_CONTROL.SET_TOT:=0; (*Reset mass flow counter*)
		Q1_CALCULETED_FLOW:=0;
		STEP := STEP+10;
	END_IF;

20: (*Continue if doors closed**************************************************************************)
	IF FLAGS.DOORS_OPEN=0 THEN
		STEP := STEP+10;
	END_IF;

30: (* Check hydraulique connexion OK*)
	Q1_DO.HYDRO_CYLINDER_BOT:=TRUE;
	Q1_DO.HYDRO_CYLINDER_TOP:=TRUE;


	STEP := STEP+10;

40: (*Continue if doors closed**************************************************************************)
	IF FLAGS.DOORS_OPEN=0 THEN
		STEP := STEP+10;
	END_IF;

50: (* Wait hydraulique connexion OK*)
	IF Q1_DI.CYLINDER_BOT_OUT AND Q1_DI.CYLINDER_TOP_OUT THEN
		STEP := STEP+10;
	END_IF;

60: (*Continue if doors closed**************************************************************************)
	IF FLAGS.DOORS_OPEN=0 THEN
		STEP := STEP+10;
	END_IF;

70: (*Close electrical connexion *)
	Q1_DO.ELECTR_CYLINDER:=TRUE;
	Q1_DO.MAX_FLOW_VALVE:=TRUE;
	STEP := STEP+10;

80: (*Continue if doors closed**************************************************************************)
	IF FLAGS.DOORS_OPEN=0 THEN
		STEP := STEP+10;
	END_IF;

90:(*Wait electrical connexion closed*)
	IF Q1_DI.POWER_CYLINDER_OUT THEN
		Start_Pump_Delay:=TRUE;
		(*Q1_DO.MAX_FLOW_VALVE:=PUMP_PARAMS.Q1_MAX_FLOW;*)
		Q1_DO.MAX_FLOW_VALVE:=TRUE;
		Q1_DO.PUMP_POWER:=TRUE;
		Q1_DO.FLOW_STOP_VALVE:=TRUE;
		Q1_DO.FLOW_STOP_BOTT:=TRUE;
		STEP := STEP+10;
	END_IF;

100: (*Continue if doors closed**************************************************************************)
	IF FLAGS.DOORS_OPEN=0 THEN
		STEP := STEP+10;
	END_IF;

110: (*Pump until end of delay*)

	(*Regulation de la pression pendant le temps d'amorcage et ne bouge plus pendant le temps de mesure*)
	(* Regulation seulement à +- 20% de la consigne et seulement après X secondes*)
	IF  Pump_Delay.ET>T#15s AND Q1_FLOWMETER_VALUES.VolumeFlow>50 THEN
				Q1_DO.MAX_FLOW_VALVE:=FALSE;
				P_ERREUR:=PUMP_PARAMS.Q1_PRESSURE_TARGET - Q1_PRESSURE_SENSOR_VALUE;
				FLAGS.MOTOR_Q1_POSITION := FLAGS.MOTOR_Q1_POSITION + REAL_TO_INT(P_ERREUR*7);(* P_ERREUR*GAIN *)
	END_IF


	IF Pump_Delay.Q THEN
		Start_Pump_Delay:=FALSE;
		Start_Measurement_Delay:=TRUE;
		Init_Mass:=Q1_FLOWMETER_VALUES.TotalMass; (*Store the mass at the beginning of the measurement*)
		STEP := STEP+10;
	END_IF;

120: (*Continue if doors closed**************************************************************************)
	IF FLAGS.DOORS_OPEN=0 THEN
		STEP := STEP+10;
	END_IF;


130: (*Measurement delay*)

	(*test*)
	IF 		(Q1_PRESSURE_SENSOR_VALUE<PUMP_PARAMS.Q1_PRESSURE_TARGET+10)
			AND (Q1_PRESSURE_SENSOR_VALUE>PUMP_PARAMS.Q1_PRESSURE_TARGET-10)
			AND Q1_FLOWMETER_VALUES.VolumeFlow>50 THEN

				P_ERREUR:=PUMP_PARAMS.Q1_PRESSURE_TARGET - Q1_PRESSURE_SENSOR_VALUE;
				FLAGS.MOTOR_Q1_POSITION := FLAGS.MOTOR_Q1_POSITION + REAL_TO_INT(P_ERREUR*7);(* P_ERREUR*GAIN *)
	END_IF
	(*end test*)

	IF Measurement_Delay.Q THEN
		Q1_CALCULETED_FLOW:=CONVERT_MASS_TO_FLOW(Q1_FLOWMETER_VALUES.TotalMass-Init_Mass, PUMP_PARAMS.Q1_MEASUREMENT_TIME); (*Convert mass to massflow*)
		Q1_DO.HYDRO_CYLINDER_BOT:=FALSE;
		Q1_DO.MAX_FLOW_VALVE:=TRUE;
		Start_Measurement_Delay:=FALSE;
		Start_FlowStop_Delay:=TRUE;
		STEP := STEP+10;
	END_IF;


140: (*Continue if doors closed**************************************************************************)
	IF FLAGS.DOORS_OPEN=0 THEN
		STEP := STEP+10;
	END_IF;


150: (*Delay before FLOWSTOP*)
	IF FlowStop_Delay.Q THEN
		Q1_DO.FLOW_STOP_VALVE:=FALSE;
		Q1_DO.MAX_FLOW_VALVE:=FALSE;
		Q1_DO.FLOW_STOP_BOTT:=FALSE;
		Q1_DO.PUMP_POWER:=FALSE;
		Start_FlowStop_Delay:=FALSE;
		bExec_DBRecordInsert1:=FALSE; (*Deactivate DB Record*)
		STEP := STEP+10;
	END_IF;


160: (*Continue if doors closed**************************************************************************)
	IF FLAGS.DOORS_OPEN=0 THEN
		STEP := STEP+10;
	END_IF;


170: (*Release electrical and hydraulic connexion*)

	Q1_DO.ELECTR_CYLINDER:=FALSE;
	Q1_DO.HYDRO_CYLINDER_TOP:=FALSE;

	STEP := STEP+10;

180: (*Continue if doors closed**************************************************************************)
	IF FLAGS.DOORS_OPEN=0 THEN
		STEP := STEP+10;
	END_IF;

190:(*Wait all cylinders IN*)
	IF Q1_DI.POWER_CYLINDER_IN AND Q1_DI.CYLINDER_TOP_IN AND Q1_DI.CYLINDER_BOT_IN THEN
		STEP := STEP+10;
	END_IF;

200: (*Continue if doors closed**************************************************************************)
	IF FLAGS.DOORS_OPEN=0 THEN
		STEP := STEP+10;
	END_IF;

210: (*Release carrier*)
	FLAGS.Q1_RELEASE_CARRIER:=TRUE;
	STEP:=STEP+10;

220: (*Continue if doors closed**************************************************************************)
	IF FLAGS.DOORS_OPEN=0 THEN
		STEP := STEP+10;
	END_IF;

230: (*Wait carrier away*)
	IF Q1_DI.WAGON_AWAY THEN
		STEP := 0;
	END_IF;



ELSE
    ;
END_CASE;

(*FBs*)
Pump_Delay(IN:= Start_Pump_Delay, PT:= PUMP_PARAMS.Q1_PUMPING_TIME);

Measurement_Delay(IN:= Start_Measurement_Delay, PT:= PUMP_PARAMS.Q1_MEASUREMENT_TIME);

FlowStop_Delay(IN:= Start_FlowStop_Delay, PT:=DRY_DELAY);

R_TRIG1(CLK:= CONVEYOR.JIG_Q1.STATUS);

PROG_STEPS.Q1_STEP:=STEP;

END_PROGRAM

// ---- GlobalTextList.TcGTLO
TEXTLIST GlobalTextList
  30 = '%.0f'
  28 = '%.1f'
  29 = '%.2f'
  22 = '%d'
  13 = '%f'
  24 = '%i'
  9 = '%s'
  8 = '%s Flag_Variables.SAFETY_IN.NOT_AUS_State'
  7 = '%s Flag_Variables.SAFETY_OUT.NOT_AUS_RESET'
  37 = 'DELTA'
  50 = 'Disable'
  5 = 'EM ACK'
  6 = 'EM Reset'
  4 = 'EM RUN'
  49 = 'Enable'
  10 = 'FIN PRODUCTION'
  3 = 'FLAGS.AUTO'
  2 = 'FLAGS.INIT_OK'
  1 = 'FLAGS.SAFETY_OK'
  53 = 'Grand Débit'
  54 = 'Petit Débit'
  36 = 'PRESSION_DEBUT'
  32 = 'Prêt à imprimer'
  25 = 'Release OPERATORS'
  41 = 'ST1'
  42 = 'ST2'
  12 = 'ST2_VACUUM'
  43 = 'ST3'
  38 = 'ST3_DELTA_P'
  35 = 'ST3_PRESSION'
  21 = 'ST4 Position moteur'
  44 = 'ST4-5'
  19 = 'ST4_CURRENT'
  34 = 'ST4_PRESSION'
  15 = 'ST4_PRESSURE'
  26 = 'ST4_Q'
  27 = 'ST4_QMAX'
  14 = 'ST4_VACUUM'
  23 = 'ST5 Position moteur'
  18 = 'ST5_CURRENT'
  17 = 'ST5_PRESSURE'
  39 = 'ST5_Q'
  40 = 'ST5_QMAX'
  16 = 'ST5_VACUUM'
  45 = 'ST6'
  20 = 'ST6_PRESSURE'
  46 = 'ST7'
  47 = 'ST8'
  31 = 'ST8 Impression OK'
  48 = 'ST9'
  51 = 'ST9 Décharge'
  52 = 'ST9 décharge'
  33 = 'STEP'
  11 = 'Test Release JIG'
  0 = 'zcxvcv'
END_TEXTLIST

// ---- VISUs/AIs.TcVIS
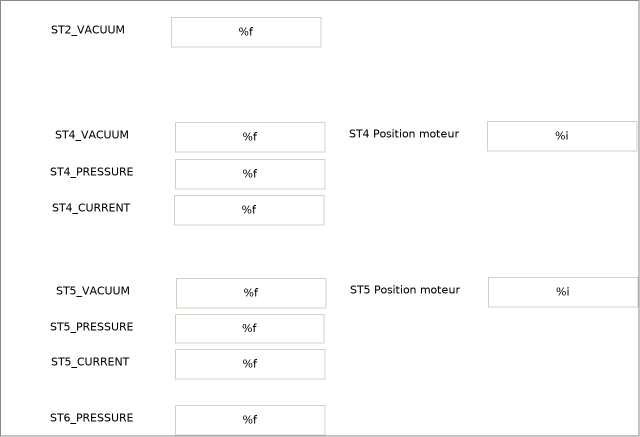
VISUALIZATION AIs  // 640x437
    Textfield (171,17 150x30), "%f", text variable: ST2_VACUUM
    Label (13,15 150x30), "ST2_VACUUM"
    Textfield (175,122 150x30), "%f", text variable: ST4_VACUUM
    Label (17,120 150x30), "ST4_VACUUM"
    Textfield (175,159 150x30), "%f", text variable: ST4_PRESSURE
    Label (17,157 150x30), "ST4_PRESSURE"
    Textfield (176,278 150x30), "%f", text variable: ST5_VACUUM
    Label (18,276 150x30), "ST5_VACUUM"
    Textfield (175,314 149x29), "%f", text variable: ST5_PRESSURE
    Label (17,312 150x30), "ST5_PRESSURE"
    Textfield (175,349 150x30), "%f", text variable: ST5_COURANT
    Label (15,347 150x30), "ST5_CURRENT"
    Textfield (174,195 150x30), "%f", text variable: ST4_COURANT
    Label (16,193 150x30), "ST4_CURRENT"
    Textfield (175,405 150x30), "%f", text variable: ST6_PRESSURE
    Label (17,403 150x30), "ST6_PRESSURE"
    Textfield (487,121 150x30), "%i", text variable: FLAGS.MOTOR_ST4_ACTUAL_POSITION
    Label (329,119 150x30), "ST4 Position moteur"
    Textfield (488,277 150x30), "%i", text variable: FLAGS.MOTOR_ST4_ACTUAL_POSITION
    Label (330,275 150x30), "ST5 Position moteur"
END_VISUALIZATION

// ---- VISUs/ST3.TcVIS
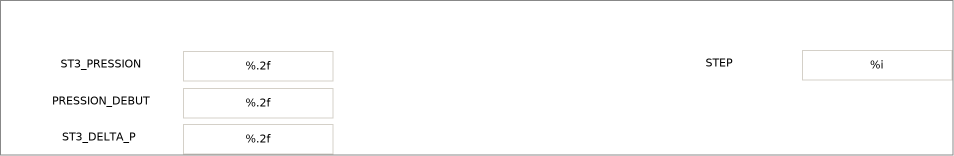
VISUALIZATION ST3  // 954x156
    Textfield (183,51 150x30), "%.2f", text variable: ST3_PRESSION
    Label (26,49 150x30), "ST3_PRESSION"
    Textfield (183,88 150x30), "%.2f", text variable: ST3_ETANCHEITE.PRESSION_DEBUT
    Label (26,86 150x30), "PRESSION_DEBUT"
    Textfield (183,124 150x30), "%.2f", text variable: ST3_DELTA_P
    Label (24,122 150x30), "ST3_DELTA_P"
    Label (644,48 150x30), "STEP"
    Textfield (802,50 150x30), "%i", text variable: IOs_Variables.PROG_STEPS.ST3
END_VISUALIZATION

// ---- VISUs/ST4.TcVIS
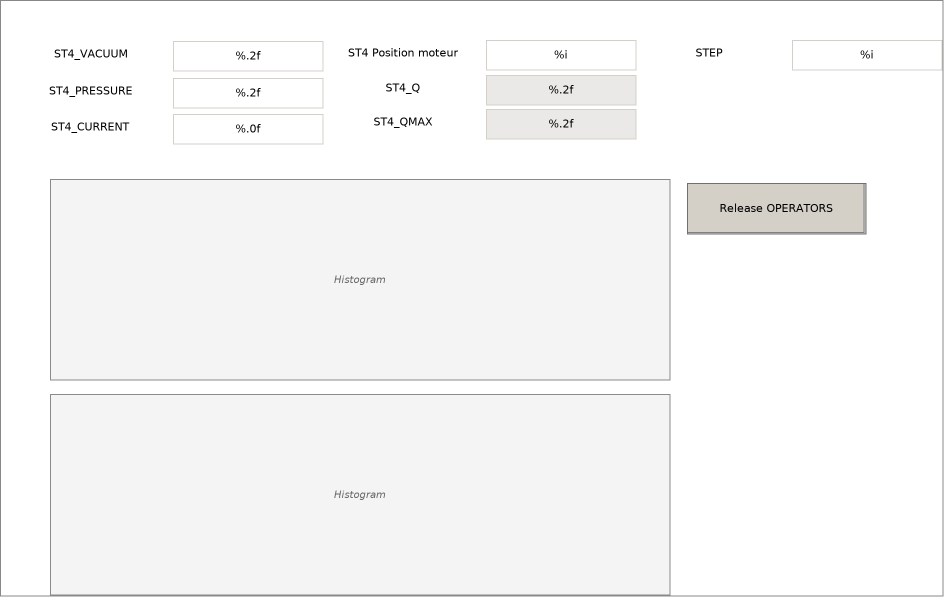
VISUALIZATION ST4  // 944x597
    Textfield (173,41 150x30), "%.2f", text variable: ST4_VACUUM
    Label (16,39 150x30), "ST4_VACUUM"
    Textfield (173,78 150x30), "%.2f", text variable: ST4_PRESSURE_FILTERED
    Label (16,76 150x30), "ST4_PRESSURE"
    Textfield (173,114 150x30), "%.0f", text variable: ST4_COURANT
    Label (15,112 150x30), "ST4_CURRENT"
    Textfield (486,40 150x30), "%i", text variable: Flag_Variables.FLAGS.MOTOR_ST4_ACTUAL_POSITION
    Label (328,38 150x30), "ST4 Position moteur"
    Textfield (486,75 150x30), "%.2f", text variable: ST4_Q
    Label (328,73 150x30), "ST4_Q"
    Textfield (486,109 150x30), "%.2f", text variable: ST4_QMAX
    Label (328,107 150x30), "ST4_QMAX"
    Histogram (50,179 620x201), scale format: %.1f, scale 20..30
        p1518820177: Flag_Variables.QMAX_ARRAY
        p102497268: Flag_Variables.QMAX_ARRAY
        p788070771: ARRAY [1..50] OF REAL
    Histogram (50,394 620x201), scale format: %.1f, scale 10..20
        p1518820177: Flag_Variables.Q_ARRAY
        p102497268: Flag_Variables.Q_ARRAY
        p788070771: ARRAY [1..50] OF REAL
    Button (687,183 179x51), "Release OPERATORS"
        tap Flag_Variables.FLAGS.DEBUG_OPERATOR
    Label (634,38 150x30), "STEP"
    Textfield (792,40 150x30), "%i", text variable: IOs_Variables.PROG_STEPS.ST4
END_VISUALIZATION

// ---- VISUs/ST5.TcVIS
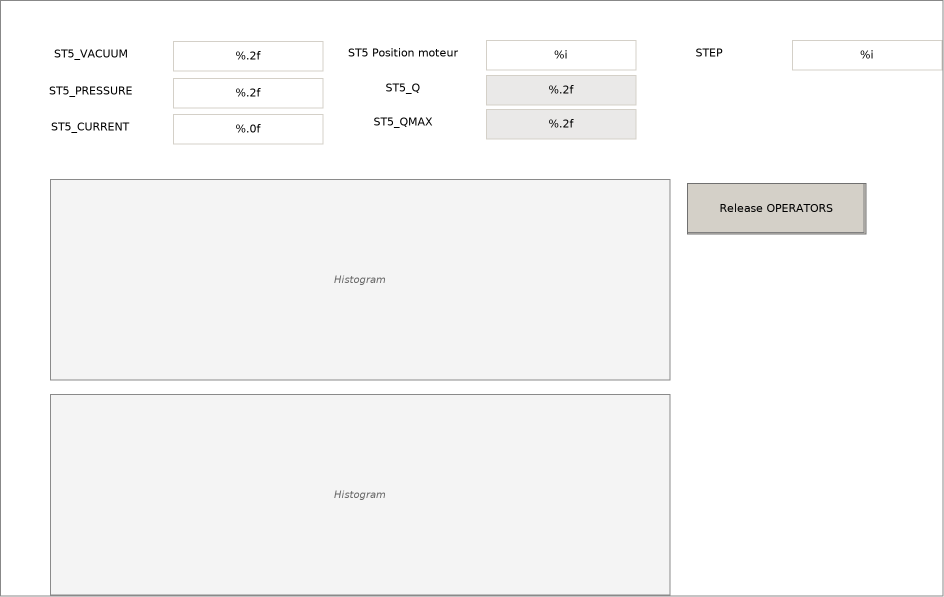
VISUALIZATION ST5  // 944x597
    Textfield (173,41 150x30), "%.2f", text variable: ST5_VACUUM
    Label (16,39 150x30), "ST5_VACUUM"
    Textfield (173,78 150x30), "%.2f", text variable: ST5_PRESSURE_FILTERED
    Label (16,76 150x30), "ST5_PRESSURE"
    Textfield (173,114 150x30), "%.0f", text variable: ST5_COURANT
    Label (15,112 150x30), "ST5_CURRENT"
    Textfield (486,40 150x30), "%i", text variable: Flag_Variables.FLAGS.MOTOR_ST5_ACTUAL_POSITION
    Label (328,38 150x30), "ST5 Position moteur"
    Textfield (486,75 150x30), "%.2f", text variable: ST5_Q
    Label (328,73 150x30), "ST5_Q"
    Textfield (486,109 150x30), "%.2f", text variable: ST5_QMAX
    Label (328,107 150x30), "ST5_QMAX"
    Histogram (50,179 620x201), scale format: %.1f, scale 20..30
        p1518820177: Flag_Variables.QMAX5_ARRAY
        p102497268: Flag_Variables.QMAX5_ARRAY
        p788070771: ARRAY [1..50] OF REAL
    Histogram (50,394 620x201), scale format: %.1f, scale 10..20
        p1518820177: Flag_Variables.Q5_ARRAY
        p102497268: Flag_Variables.Q5_ARRAY
        p788070771: ARRAY [1..50] OF REAL
    Button (687,183 179x51), "Release OPERATORS"
        tap Flag_Variables.FLAGS.DEBUG_OPERATOR
    Label (634,38 150x30), "STEP"
    Textfield (792,40 150x30), "%i", text variable: IOs_Variables.PROG_STEPS.ST5
END_VISUALIZATION

// ---- VISUs/Visualization.TcVIS
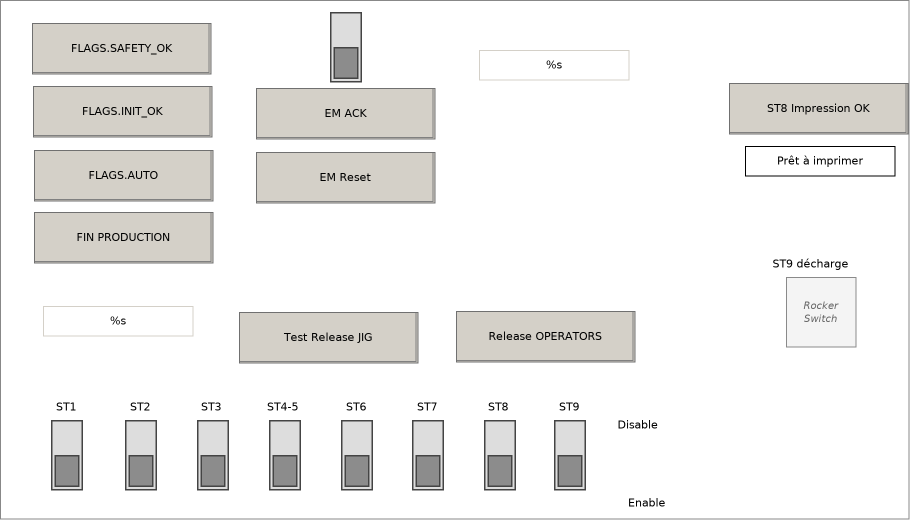
VISUALIZATION Visualization  // 910x520
    Button (32,23 179x51), "FLAGS.SAFETY_OK"
        toggle Flag_Variables.FLAGS.SAFETY_OK
    Button (33,86 179x51), "FLAGS.INIT_OK"
        toggle Flag_Variables.FLAGS.INIT_OK
    Button (34,150 179x51), "FLAGS.AUTO"
        toggle Flag_Variables.FLAGS.AUTO
    Button (256,88 179x51), "EM ACK"
        tap Flag_Variables.SAFETY_OUT.NOT_AUS_ErrAck
    Button (256,152 179x51), "EM Reset"
        tap Flag_Variables.SAFETY_OUT.NOT_AUS_RESET
    DipSwitch (311,12 70x70), variable: Flag_Variables.SAFETY_OUT.NOT_AUS_RUN, behaviour: TOGGLE, style: Switch-DipSwitch-Gray
    Textfield (479,50 150x30), "%s", text variable: Flag_Variables.SAFETY_IN.NOT_AUS_State
    Textfield (43,306 150x30), "%s", text variable: GEMMA.STEP
    Button (34,212 179x51), "FIN PRODUCTION"
        tap GEMMA.F2_END
    Button (239,312 179x51), "Test Release JIG"
        tap CONVEYOR.TEST_RELEASE
    Button (456,311 179x51), "Release OPERATORS"
        tap Flag_Variables.FLAGS.DEBUG_OPERATOR
    Button (729,83 179x51), "ST8 Impression OK"
        tap IOs_Variables.ST8_IMPRESSION_OK
    Rectangle (745,146 150x30), "Prêt à imprimer", colour toggle: IOs_Variables.ST8_PRET_A_IMPRIMER
    DipSwitch (32,420 70x70), variable: ST1_JIG_DISABLED, behaviour: TOGGLE, style: Switch-DipSwitch-Gray
    DipSwitch (106,420 70x70), variable: ST2_JIG_DISABLED, behaviour: TOGGLE, style: Switch-DipSwitch-Gray
    DipSwitch (178,420 70x70), variable: ST3_JIG_DISABLED, behaviour: TOGGLE, style: Switch-DipSwitch-Gray
    DipSwitch (250,420 70x70), variable: ST4_5_JIG_DISABLED, behaviour: TOGGLE, style: Switch-DipSwitch-Gray
    DipSwitch (322,420 70x70), variable: ST6_JIG_DISABLED, behaviour: TOGGLE, style: Switch-DipSwitch-Gray
    DipSwitch (393,420 70x70), variable: ST7_JIG_DISABLED, behaviour: TOGGLE, style: Switch-DipSwitch-Gray
    DipSwitch (465,420 70x70), variable: ST8_JIG_DISABLED, behaviour: TOGGLE, style: Switch-DipSwitch-Gray
    DipSwitch (535,420 70x70), variable: ST9_JIG_DISABLED, behaviour: TOGGLE, style: Switch-DipSwitch-Gray
    Label (48,392 37x30), "ST1"
    Label (122,392 37x30), "ST2"
    Label (193,392 37x30), "ST3"
    Label (256,392 54x30), "ST4-5"
    Label (338,392 37x30), "ST6"
    Label (409,392 37x30), "ST7"
    Label (480,392 37x30), "ST8"
    Label (551,392 37x30), "ST9"
    Label (743,249 135x30), "ST9 décharge"
    Label (602,410 72x30), "Disable"
    RockerSwitch (786,277 70x70), variable: ST9_DECHARGE, behaviour: TOGGLE, style: Switch-RockerSwitch-Gray
    Label (611,488 72x30), "Enable"
END_VISUALIZATION
